KUKA KRL program: MyProgram_287().src

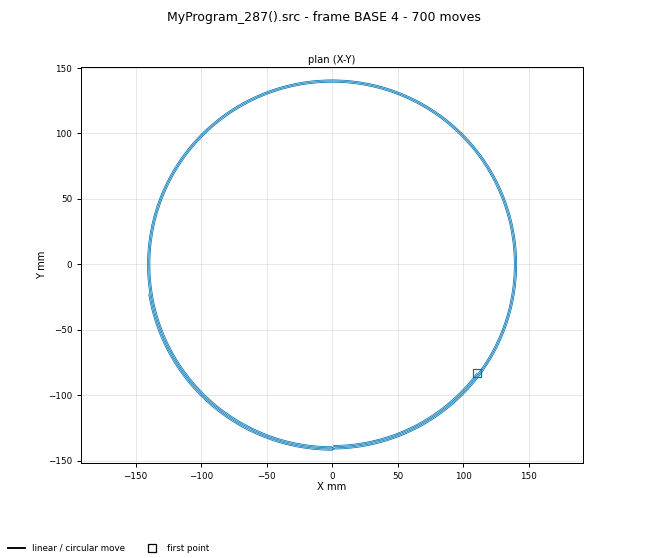
[picture p0: tool path of MyProgram_287().src in frame BASE 4, 700 of 700 moves have a stored position in this frame; points joined in program order, loops and branches not executed]
&ACCESS RVP
&REL 1
&PARAM TEMPLATE = C:\KRC\Roboter\Template\vorgabe
&PARAM EDITMASK = *
DEF MyProgram_287()
; ---- Setting reference (Base) ----
$BASE = BASE_DATA[4]

; --------------------------
; ---- Setting tool (TCP) ----
$TOOL = TOOL_DATA[3]
; --------------------------

$VEL.CP = VEL_APROX_PRINT
Startdeposition()
$VEL.CP = VEL_PRINT
LIN {X 110.6331,Y -82.8867,Z 175,A -34.5212,B 7.5627,C 0.3463,E1 7.6986,E2 486.4179} C_DIS
LIN {X 107.2416,Y -87.2299,Z 175,A -36.9213,B 7.5624,C 0.3539,E1 7.6944,E2 488.8351} C_DIS
LIN {X 102.8768,Y -92.3369,Z 175,A -39.3505,B 7.5624,C 0.3533,E1 7.69,E2 491.2213} C_DIS
LIN {X 98.1366,Y -97.3598,Z 175,A -42.4182,B 7.5619,C 0.3634,E1 7.6841,E2 494.3184} C_DIS
LIN {X 93.1713,Y -102.1223,Z 175,A -45.0279,B 7.5619,C 0.3647,E1 7.6789,E2 496.8996} C_DIS
LIN {X 87.5657,Y -106.9672,Z 175,A -48.9682,B 7.5608,C 0.3871,E1 7.6702,E2 500.9543} C_DIS
LIN {X 82.9444,Y -110.5898,Z 175,A -50.7968,B 7.5611,C 0.3802,E1 7.6663,E2 502.7077} C_DIS
LIN {X 78.2909,Y -113.9309,Z 175,A -53.0648,B 7.561,C 0.3823,E1 7.6611,E2 504.9642} C_DIS
LIN {X 74.3872,Y -116.5173,Z 175,A -54.9775,B 7.5609,C 0.3851,E1 7.6567,E2 506.8749} C_DIS
LIN {X 69.3615,Y -119.5773,Z 175,A -57.3901,B 7.5607,C 0.3884,E1 7.6509,E2 509.2862} C_DIS
LIN {X 65.5707,Y -121.6973,Z 175,A -59.228,B 7.5605,C 0.3918,E1 7.6464,E2 511.1304} C_DIS
LIN {X 61.8336,Y -123.6379,Z 175,A -60.9301,B 7.5605,C 0.3934,E1 7.6421,E2 512.8284} C_DIS
LIN {X 58.7912,Y -125.1139,Z 175,A -62.3873,B 7.5603,C 0.3963,E1 7.6385,E2 514.2939} C_DIS
LIN {X 53.8239,Y -127.3284,Z 175,A -64.525,B 7.5603,C 0.397,E1 7.633,E2 516.4183} C_DIS
LIN {X 49.8285,Y -128.9433,Z 175,A -66.4746,B 7.56,C 0.4021,E1 7.6279,E2 518.3903} C_DIS
LIN {X 45.7126,Y -130.4598,Z 175,A -68.0713,B 7.56,C 0.4001,E1 7.6238,E2 519.9599} C_DIS
LIN {X 41.2974,Y -131.9257,Z 175,A -70.0623,B 7.56,C 0.4031,E1 7.6184,E2 521.9604} C_DIS
LIN {X 37.6293,Y -133.0166,Z 175,A -71.3805,B 7.5601,C 0.3998,E1 7.615,E2 523.2451} C_DIS
LIN {X 34.2562,Y -133.9246,Z 175,A -73.2007,B 7.5597,C 0.4076,E1 7.6099,E2 525.1143} C_DIS
LIN {X 29.37,Y -135.0803,Z 175,A -75.02,B 7.5599,C 0.4046,E1 7.6051,E2 526.9012} C_DIS
LIN {X 26.0323,Y -135.7629,Z 175,A -76.4292,B 7.5599,C 0.4055,E1 7.6012,E2 528.3109} C_DIS
LIN {X 22.9559,Y -136.317,Z 175,A -78.4903,B 7.559,C 0.4196,E1 7.5953,E2 530.471} C_DIS
LIN {X 16.9955,Y -137.189,Z 175,A -80.2487,B 7.5597,C 0.408,E1 7.5907,E2 532.1364} C_DIS
LIN {X 13.2679,Y -137.5982,Z 175,A -81.6417,B 7.5597,C 0.4059,E1 7.5868,E2 533.5094} C_DIS
LIN {X 10.1361,Y -137.8643,Z 175,A -83.1514,B 7.5596,C 0.4099,E1 7.5826,E2 535.0465} C_DIS
LIN {X 5.4762,Y -138.128,Z 175,A -85.0409,B 7.5596,C 0.4096,E1 7.5773,E2 536.9311} C_DIS
LIN {X 1.0216,Y -138.2328,Z 175,A -86.8303,B 7.5596,C 0.409,E1 7.5723,E2 538.714} C_DIS
Enddeposition()
LIN {X 1.0216,Y -138.2328,Z 175,A -86.8303,B 7.5596,C 0.409,E1 7.5723,E2 538.714} C_DIS
Startdeposition()
$VEL.CP = VEL_PRINT
LIN {X 1.4201,Y -139.1373,Z 175,A -85.8495,B 7.508,C 0.3996,E1 7.5232,E2 537.6751} C_DIS
LIN {X 5.8285,Y -139.0214,Z 175,A -84.1991,B 7.5079,C 0.4021,E1 7.5277,E2 536.0455} C_DIS
LIN {X 9.2409,Y -138.8374,Z 175,A -82.6419,B 7.508,C 0.399,E1 7.5321,E2 534.4679} C_DIS
LIN {X 13.2856,Y -138.5071,Z 175,A -81.1056,B 7.508,C 0.4008,E1 7.5364,E2 532.9483} C_DIS
LIN {X 16.7511,Y -138.1311,Z 175,A -79.5636,B 7.508,C 0.3982,E1 7.5407,E2 531.3915} C_DIS
LIN {X 23.3229,Y -137.1748,Z 175,A -76.3997,B 7.5086,C 0.389,E1 7.5496,E2 528.1692} C_DIS
LIN {X 27.9525,Y -136.3062,Z 175,A -74.9929,B 7.5081,C 0.3973,E1 7.5532,E2 526.8316} C_DIS
LIN {X 35.5217,Y -134.5325,Z 175,A -72.0188,B 7.5081,C 0.3989,E1 7.5613,E2 523.8855} C_DIS
LIN {X 37.6917,Y -133.9405,Z 175,A -70.9319,B 7.5082,C 0.3951,E1 7.5642,E2 522.7769} C_DIS
LIN {X 41.1973,Y -132.9048,Z 175,A -69.4338,B 7.5083,C 0.3938,E1 7.5682,E2 521.2786} C_DIS
LIN {X 44.3172,Y -131.8968,Z 175,A -67.7638,B 7.5087,C 0.3866,E1 7.5728,E2 519.5654} C_DIS
LIN {X 47.5641,Y -130.761,Z 175,A -66.6566,B 7.5085,C 0.3908,E1 7.5756,E2 518.4981} C_DIS
LIN {X 51.0181,Y -129.4534,Z 175,A -65.0237,B 7.5087,C 0.3869,E1 7.5799,E2 516.8493} C_DIS
LIN {X 56.479,Y -127.1647,Z 175,A -62.7406,B 7.5087,C 0.3868,E1 7.5857,E2 514.5847} C_DIS
LIN {X 58.8003,Y -126.1084,Z 175,A -61.674,B 7.5087,C 0.3851,E1 7.5884,E2 513.5151} C_DIS
LIN {X 62.3508,Y -124.3934,Z 175,A -60.0875,B 7.5088,C 0.3836,E1 7.5924,E2 511.9322} C_DIS
LIN {X 65.2663,Y -122.8874,Z 175,A -58.7004,B 7.509,C 0.381,E1 7.5958,E2 510.5393} C_DIS
LIN {X 69.1818,Y -120.7274,Z 175,A -56.0217,B 7.5099,C 0.3623,E1 7.6026,E2 507.7481} C_DIS
LIN {X 74.9621,Y -117.2256,Z 175,A -54.2838,B 7.5091,C 0.3777,E1 7.6064,E2 506.1462} C_DIS
LIN {X 77.8365,Y -115.3373,Z 175,A -52.1354,B 7.5099,C 0.3613,E1 7.6116,E2 503.8999} C_DIS
LIN {X 82.166,Y -112.2942,Z 175,A -50.8362,B 7.5093,C 0.3743,E1 7.6143,E2 502.715} C_DIS
LIN {X 85.7474,Y -109.5838,Z 175,A -48.8324,B 7.5096,C 0.368,E1 7.6188,E2 500.6893} C_DIS
LIN {X 88.6836,Y -107.2212,Z 175,A -46.6577,B 7.5103,C 0.353,E1 7.6236,E2 498.4309} C_DIS
LIN {X 92.5552,Y -103.8977,Z 175,A -45.0634,B 7.5101,C 0.3586,E1 7.6268,E2 496.9018} C_DIS
LIN {X 95.9429,Y -100.7779,Z 175,A -43.2164,B 7.5102,C 0.3557,E1 7.6306,E2 495.0595} C_DIS
LIN {X 99.1505,Y -97.6238,Z 175,A -40.9161,B 7.5108,C 0.343,E1 7.6352,E2 492.6983} C_DIS
LIN {X 102.5453,Y -94.0513,Z 175,A -39.4326,B 7.5105,C 0.3493,E1 7.6379,E2 491.2849} C_DIS
LIN {X 106.3749,Y -89.6976,Z 175,A -37.3257,B 7.5105,C 0.3494,E1 7.6417,E2 489.2125} C_DIS
LIN {X 111.1691,Y -83.6817,Z 175,A -33.9616,B 7.511,C 0.3383,E1 7.6476,E2 485.8198} C_DIS
LIN {X 113.8489,Y -79.9979,Z 175,A -32.0815,B 7.5112,C 0.3337,E1 7.6506,E2 483.9372} C_DIS
LIN {X 116.2575,Y -76.455,Z 175,A -30.3464,B 7.5114,C 0.3299,E1 7.6533,E2 482.2042} C_DIS
LIN {X 119.2524,Y -71.6949,Z 175,A -28.1739,B 7.5115,C 0.327,E1 7.6565,E2 480.0482} C_DIS
LIN {X 121.1264,Y -68.4812,Z 175,A -26.5315,B 7.5118,C 0.3209,E1 7.6588,E2 478.3899} C_DIS
LIN {X 123.125,Y -64.814,Z 175,A -24.7076,B 7.512,C 0.3143,E1 7.6612,E2 476.5506} C_DIS
LIN {X 124.5929,Y -61.9468,Z 175,A -23.8146,B 7.5118,C 0.3195,E1 7.6622,E2 475.713} C_DIS
LIN {X 128.0502,Y -54.4463,Z 175,A -20.2779,B 7.5123,C 0.3078,E1 7.6664,E2 472.1556} C_DIS
LIN {X 129.844,Y -50.0134,Z 175,A -18.3416,B 7.5125,C 0.3031,E1 7.6683,E2 470.2216} C_DIS
LIN {X 130.9587,Y -47.0157,Z 175,A -17.0459,B 7.5126,C 0.2999,E1 7.6696,E2 468.9273} C_DIS
LIN {X 132.1846,Y -43.4529,Z 175,A -15.5767,B 7.5127,C 0.2973,E1 7.6709,E2 467.4674} C_DIS
LIN {X 133.6756,Y -38.6231,Z 175,A -13.2766,B 7.5131,C 0.2871,E1 7.6727,E2 465.1368} C_DIS
LIN {X 134.9715,Y -33.8161,Z 175,A -11.506,B 7.5131,C 0.287,E1 7.6739,E2 463.4006} C_DIS
LIN {X 135.7081,Y -30.7257,Z 175,A -10.2142,B 7.5133,C 0.2836,E1 7.6747,E2 462.1097} C_DIS
LIN {X 137.0688,Y -23.9412,Z 175,A -7.6666,B 7.5133,C 0.2816,E1 7.6761,E2 459.5988} C_DIS
LIN {X 137.6462,Y -20.3642,Z 175,A -6.0341,B 7.5136,C 0.2745,E1 7.6768,E2 457.9467} C_DIS
LIN {X 138.0565,Y -17.3679,Z 175,A -4.6261,B 7.5138,C 0.2677,E1 7.6773,E2 456.5165} C_DIS
LIN {X 138.7792,Y -10.0537,Z 175,A -1.8474,B 7.514,C 0.264,E1 7.678,E2 453.7672} C_DIS
LIN {X 138.9752,Y -6.8315,Z 175,A -0.4575,B 7.5141,C 0.2589,E1 7.6782,E2 452.3683} C_DIS
LIN {X 139.1026,Y -3.3845,Z 175,A 0.8979,B 7.5142,C 0.2561,E1 7.6784,E2 451.0201} C_DIS
LIN {X 139.1434,Y -0.4634,Z 175,A 2.037,B 7.5143,C 0.254,E1 7.6784,E2 449.8883} C_DIS
LIN {X 139.1107,Y 3.0949,Z 175,A 3.7076,B 7.5146,C 0.2456,E1 7.6784,E2 448.1898} C_DIS
LIN {X 138.8806,Y 8.5391,Z 175,A 5.8033,B 7.5147,C 0.2421,E1 7.678,E2 446.1113} C_DIS
LIN {X 138.5278,Y 13.0704,Z 175,A 8.0872,B 7.5151,C 0.2285,E1 7.6774,E2 443.7724} C_DIS
LIN {X 138.0155,Y 17.6805,Z 175,A 10.4809,B 7.5156,C 0.2133,E1 7.6765,E2 441.3139} C_DIS
LIN {X 136.852,Y 25.1523,Z 175,A 12.4644,B 7.5152,C 0.2272,E1 7.6757,E2 439.4752} C_DIS
LIN {X 135.5461,Y 31.4349,Z 175,A 15.0748,B 7.5154,C 0.2204,E1 7.6741,E2 436.867} C_DIS
LIN {X 134.6874,Y 34.9355,Z 175,A 16.5343,B 7.5154,C 0.2168,E1 7.6731,E2 435.4096} C_DIS
LIN {X 133.9536,Y 37.6448,Z 175,A 17.668,B 7.5155,C 0.214,E1 7.6723,E2 434.278} C_DIS
LIN {X 132.9674,Y 40.9925,Z 175,A 19.089,B 7.5157,C 0.2104,E1 7.6711,E2 432.8579} C_DIS
LIN {X 132.0076,Y 43.9844,Z 175,A 20.3873,B 7.5157,C 0.2068,E1 7.67,E2 431.5582} C_DIS
LIN {X 130.8447,Y 47.332,Z 175,A 21.8394,B 7.5159,C 0.203,E1 7.6686,E2 430.1061} C_DIS
LIN {X 129.5562,Y 50.7537,Z 175,A 23.2485,B 7.5159,C 0.2008,E1 7.6672,E2 428.7085} C_DIS
LIN {X 127.2737,Y 56.2354,Z 175,A 25.6984,B 7.5161,C 0.1943,E1 7.6646,E2 426.2565} C_DIS
LIN {X 125.0302,Y 61.0602,Z 175,A 27.7239,B 7.5161,C 0.1919,E1 7.6622,E2 424.2509} C_DIS
LIN {X 123.8823,Y 63.3549,Z 175,A 28.903,B 7.5163,C 0.1868,E1 7.6607,E2 423.0555} C_DIS
LIN {X 121.9898,Y 66.9311,Z 175,A 30.8976,B 7.5165,C 0.1762,E1 7.658,E2 421.018} C_DIS
LIN {X 120.1169,Y 70.2345,Z 175,A 32.4748,B 7.5166,C 0.172,E1 7.6557,E2 419.4382} C_DIS
LIN {X 117.9562,Y 73.808,Z 175,A 33.7508,B 7.5166,C 0.1765,E1 7.6539,E2 418.2183} C_DIS
LIN {X 115.7509,Y 77.2197,Z 175,A 35.2951,B 7.5166,C 0.175,E1 7.6516,E2 416.6896} C_DIS
LIN {X 113.7648,Y 80.1171,Z 175,A 36.9071,B 7.5167,C 0.1684,E1 7.649,E2 415.0558} C_DIS
LIN {X 110.9929,Y 83.9151,Z 175,A 39.2311,B 7.517,C 0.1565,E1 7.645,E2 412.6813} C_DIS
LIN {X 108.1615,Y 87.5345,Z 175,A 40.6057,B 7.5168,C 0.1622,E1 7.6427,E2 411.3722} C_DIS
LIN {X 105.5905,Y 90.6194,Z 175,A 42.3243,B 7.5169,C 0.1573,E1 7.6396,E2 409.6448} C_DIS
LIN {X 99.9105,Y 96.8455,Z 175,A 45.3488,B 7.5169,C 0.1585,E1 7.634,E2 406.6759} C_DIS
LIN {X 96.1312,Y 100.5973,Z 175,A 47.9075,B 7.5171,C 0.1472,E1 7.6288,E2 404.0703} C_DIS
LIN {X 93.3186,Y 103.2126,Z 175,A 49.4134,B 7.5171,C 0.1456,E1 7.6257,E2 402.5736} C_DIS
LIN {X 91.2332,Y 105.0608,Z 175,A 50.5802,B 7.5172,C 0.1431,E1 7.6233,E2 401.4041} C_DIS
LIN {X 87.8054,Y 107.942,Z 175,A 52.4091,B 7.5172,C 0.14,E1 7.6193,E2 399.5768} C_DIS
LIN {X 84.2147,Y 110.7664,Z 175,A 54.2717,B 7.5173,C 0.137,E1 7.6152,E2 397.7161} C_DIS
LIN {X 80.5882,Y 113.4322,Z 175,A 56.2153,B 7.5174,C 0.1323,E1 7.6108,E2 395.7609} C_DIS
LIN {X 75.6902,Y 116.7569,Z 175,A 58.3095,B 7.5174,C 0.1347,E1 7.606,E2 393.7099} C_DIS
LIN {X 72.5843,Y 118.7128,Z 175,A 59.9518,B 7.5174,C 0.13,E1 7.6021,E2 392.051} C_DIS
LIN {X 68.9617,Y 120.853,Z 175,A 61.7195,B 7.5175,C 0.1269,E1 7.5978,E2 390.2788} C_DIS
LIN {X 65.0323,Y 123.0104,Z 175,A 64.5964,B 7.5178,C 0.1057,E1 7.5904,E2 387.2703} C_DIS
LIN {X 57.7968,Y 126.5724,Z 175,A 66.851,B 7.5176,C 0.1209,E1 7.585,E2 385.152} C_DIS
LIN {X 51.8404,Y 129.1249,Z 175,A 69.4055,B 7.5176,C 0.12,E1 7.5785,E2 382.6122} C_DIS
LIN {X 48.426,Y 130.4443,Z 175,A 70.8827,B 7.5176,C 0.119,E1 7.5746,E2 381.139} C_DIS
LIN {X 44.9713,Y 131.6762,Z 175,A 72.3636,B 7.5176,C 0.1181,E1 7.5707,E2 379.6621} C_DIS
LIN {X 41.8074,Y 132.7143,Z 175,A 73.7259,B 7.5176,C 0.117,E1 7.5671,E2 378.301} C_DIS
LIN {X 38.8998,Y 133.5946,Z 175,A 75.0449,B 7.5177,C 0.1148,E1 7.5635,E2 376.9736} C_DIS
LIN {X 35.5899,Y 134.5143,Z 175,A 76.4451,B 7.5177,C 0.114,E1 7.5598,E2 375.5756} C_DIS
LIN {X 31.1855,Y 135.603,Z 175,A 78.2197,B 7.5177,C 0.1144,E1 7.555,E2 373.8132} C_DIS
LIN {X 24.6353,Y 136.9446,Z 175,A 80.7589,B 7.5177,C 0.1165,E1 7.5481,E2 371.3017} C_DIS
LIN {X 17.9569,Y 137.9793,Z 175,A 83.8373,B 7.5177,C 0.1103,E1 7.5395,E2 368.1873} C_DIS
LIN {X 13.5162,Y 138.485,Z 175,A 85.6921,B 7.5177,C 0.1095,E1 7.5344,E2 366.3314} C_DIS
LIN {X 9.3418,Y 138.8311,Z 175,A 87.5643,B 7.5178,C 0.1067,E1 7.5291,E2 364.4414} C_DIS
LIN {X 4.7477,Y 139.0636,Z 175,A 89.3336,B 7.5178,C 0.1085,E1 7.5242,E2 362.6886} C_DIS
LIN {X 0.3427,Y 139.1432,Z 175,A 91.0081,B 7.5178,C 0.1108,E1 7.5196,E2 361.0324} C_DIS
LIN {X -3.1295,Y 139.1097,Z 175,A 92.5251,B 7.5178,C 0.1094,E1 7.5153,E2 359.5052} C_DIS
LIN {X -9.7529,Y 138.8012,Z 175,A 95.0699,B 7.5178,C 0.1129,E1 7.5083,E2 356.985} C_DIS
LIN {X -16.5387,Y 138.1564,Z 175,A 98.0944,B 7.5178,C 0.1102,E1 7.4998,E2 353.9349} C_DIS
LIN {X -23.5222,Y 137.1415,Z 175,A 100.901,B 7.5178,C 0.113,E1 7.4921,E2 351.1425} C_DIS
LIN {X -26.4114,Y 136.6134,Z 175,A 102.1282,B 7.5178,C 0.1134,E1 7.4887,E2 349.9138} C_DIS
LIN {X -29.4419,Y 135.9921,Z 175,A 103.4486,B 7.5178,C 0.1134,E1 7.4851,E2 348.5883} C_DIS
LIN {X -33.1224,Y 135.1438,Z 175,A 105.0333,B 7.5178,C 0.114,E1 7.4808,E2 347.001} C_DIS
LIN {X -37.9549,Y 133.8668,Z 175,A 107.0155,B 7.5177,C 0.1167,E1 7.4755,E2 345.0297} C_DIS
LIN {X -41.1039,Y 132.9334,Z 175,A 108.3808,B 7.5177,C 0.1177,E1 7.4718,E2 343.6636} C_DIS
LIN {X -44.4666,Y 131.8471,Z 175,A 110.1098,B 7.5177,C 0.1147,E1 7.4671,E2 341.9013} C_DIS
LIN {X -50.2139,Y 129.7661,Z 175,A 112.5513,B 7.5177,C 0.1184,E1 7.4608,E2 339.4711} C_DIS
LIN {X -53.8552,Y 128.2977,Z 175,A 114.0667,B 7.5176,C 0.1218,E1 7.4569,E2 337.9696} C_DIS
LIN {X -57.3649,Y 126.7685,Z 175,A 116.1592,B 7.5176,C 0.1158,E1 7.4514,E2 335.8134} C_DIS
LIN {X -61.3669,Y 124.8789,Z 175,A 117.245,B 7.5175,C 0.1292,E1 7.4489,E2 334.8216} C_DIS
LIN {X -65.5803,Y 122.7212,Z 175,A 119.5789,B 7.5175,C 0.1261,E1 7.443,E2 332.4412} C_DIS
LIN {X -71.8801,Y 119.1404,Z 175,A 122.4019,B 7.5175,C 0.1328,E1 7.4363,E2 329.6409} C_DIS
LIN {X -75.9748,Y 116.5721,Z 175,A 124.5763,B 7.5175,C 0.1332,E1 7.4311,E2 327.445} C_DIS
LIN {X -79.8148,Y 113.9778,Z 175,A 126.5319,B 7.5174,C 0.1356,E1 7.4266,E2 325.4852} C_DIS
LIN {X -86.6506,Y 108.8707,Z 175,A 129.8564,B 7.5172,C 0.1445,E1 7.4192,E2 322.1877} C_DIS
LIN {X -89.3495,Y 106.6669,Z 175,A 131.5183,B 7.5172,C 0.1439,E1 7.4156,E2 320.4985} C_DIS
LIN {X -93.9561,Y 102.6328,Z 175,A 134.4308,B 7.5172,C 0.1431,E1 7.4094,E2 317.539} C_DIS
LIN {X -97.0129,Y 99.7485,Z 175,A 135.5603,B 7.517,C 0.1552,E1 7.4073,E2 316.4868} C_DIS
LIN {X -99.059,Y 97.7171,Z 175,A 137.0419,B 7.517,C 0.1534,E1 7.4043,E2 314.9693} C_DIS
LIN {X -103.493,Y 93.0077,Z 175,A 139.8811,B 7.517,C 0.1566,E1 7.3989,E2 312.1105} C_DIS
LIN {X -106.4377,Y 89.6228,Z 175,A 141.6227,B 7.5168,C 0.1622,E1 7.3958,E2 310.3841} C_DIS
LIN {X -109.2153,Y 86.2165,Z 175,A 143.5593,B 7.5168,C 0.1645,E1 7.3924,E2 308.4332} C_DIS
LIN {X -111.958,Y 82.6236,Z 175,A 145.2151,B 7.5166,C 0.1717,E1 7.3897,E2 306.8051} C_DIS
LIN {X -114.3086,Y 79.3394,Z 175,A 146.9862,B 7.5166,C 0.1741,E1 7.3868,E2 305.022} C_DIS
LIN {X -116.6391,Y 75.8715,Z 175,A 149.1485,B 7.5166,C 0.1721,E1 7.3834,E2 302.8054} C_DIS
LIN {X -118.9143,Y 72.254,Z 175,A 150.5098,B 7.5164,C 0.182,E1 7.3815,E2 301.4963} C_DIS
LIN {X -121.0516,Y 68.6136,Z 175,A 152.4285,B 7.5164,C 0.1839,E1 7.3788,E2 299.5564} C_DIS
LIN {X -123.3582,Y 64.3699,Z 175,A 154.2955,B 7.5162,C 0.1906,E1 7.3764,E2 297.7067} C_DIS
LIN {X -125.9505,Y 59.1418,Z 175,A 156.6895,B 7.516,C 0.197,E1 7.3734,E2 295.3164} C_DIS
LIN {X -127.1149,Y 56.5904,Z 175,A 157.8993,B 7.516,C 0.1993,E1 7.372,E2 294.1006} C_DIS
LIN {X -128.6045,Y 53.1206,Z 175,A 159.5168,B 7.5159,C 0.2026,E1 7.3703,E2 292.4767} C_DIS
LIN {X -129.7693,Y 50.2057,Z 175,A 160.8193,B 7.5158,C 0.2059,E1 7.369,E2 291.1742} C_DIS
LIN {X -131.0451,Y 46.7761,Z 175,A 162.3069,B 7.5157,C 0.2103,E1 7.3675,E2 289.6905} C_DIS
LIN {X -132.1799,Y 43.4669,Z 175,A 163.7712,B 7.5156,C 0.2139,E1 7.3662,E2 288.2247} C_DIS
LIN {X -133.1893,Y 40.2675,Z 175,A 165.176,B 7.5155,C 0.2174,E1 7.3651,E2 286.8181} C_DIS
LIN {X -134.0766,Y 37.2047,Z 175,A 166.4876,B 7.5153,C 0.2211,E1 7.3641,E2 285.5079} C_DIS
LIN {X -134.934,Y 33.9641,Z 175,A 167.9478,B 7.5153,C 0.2238,E1 7.3631,E2 284.039} C_DIS
LIN {X -135.7747,Y 30.434,Z 175,A 169.4504,B 7.5151,C 0.2279,E1 7.3621,E2 282.5367} C_DIS
LIN {X -137.0284,Y 24.1669,Z 175,A 172.0912,B 7.5149,C 0.2353,E1 7.3607,E2 279.8973} C_DIS
LIN {X -137.5307,Y 21.1194,Z 175,A 173.4536,B 7.5149,C 0.2377,E1 7.3601,E2 278.5245} C_DIS
LIN {X -138.0249,Y 17.6089,Z 175,A 174.9348,B 7.5147,C 0.2416,E1 7.3596,E2 277.042} C_DIS
LIN {X -138.6421,Y 11.794,Z 175,A 177.964,B 7.5147,C 0.24,E1 7.3588,E2 273.9355} C_DIS
LIN {X -138.9674,Y 6.9865,Z 175,A 179.1814,B 7.5142,C 0.2562,E1 7.3586,E2 272.8179} C_DIS
LIN {X -139.0886,Y 3.8883,Z 175,A -179.2932,B 7.5142,C 0.2565,E1 7.3584,E2 271.2621} C_DIS
LIN {X -139.1227,Y -2.3738,Z 175,A -176.2102,B 7.5142,C 0.257,E1 7.3584,E2 268.1167} C_DIS
LIN {X -138.9902,Y -6.5331,Z 175,A -174.9194,B 7.5138,C 0.2677,E1 7.3586,E2 266.8816} C_DIS
LIN {X -138.7817,Y -10.0191,Z 175,A -173.4204,B 7.5138,C 0.271,E1 7.3589,E2 265.376} C_DIS
LIN {X -137.9589,Y -18.1126,Z 175,A -170.291,B 7.5133,C 0.2836,E1 7.3598,E2 262.2777} C_DIS
LIN {X -137.5237,Y -21.1652,Z 175,A -168.7207,B 7.5133,C 0.2831,E1 7.3605,E2 260.6699} C_DIS
LIN {X -136.9491,Y -24.6097,Z 175,A -167.2575,B 7.5131,C 0.2868,E1 7.3612,E2 259.2047} C_DIS
LIN {X -136.3006,Y -27.9804,Z 175,A -165.787,B 7.5131,C 0.29,E1 7.362,E2 257.7279} C_DIS
LIN {X -135.5939,Y -31.2254,Z 175,A -164.4008,B 7.5129,C 0.2936,E1 7.3628,E2 256.3404} C_DIS
LIN {X -134.5408,Y -35.4905,Z 175,A -162.5242,B 7.5127,C 0.2977,E1 7.3641,E2 254.4564} C_DIS
LIN {X -133.5579,Y -39.0249,Z 175,A -161.0415,B 7.5125,C 0.3022,E1 7.3652,E2 252.9783} C_DIS
LIN {X -132.543,Y -42.3438,Z 175,A -159.5616,B 7.5125,C 0.3054,E1 7.3665,E2 251.4929} C_DIS
LIN {X -131.4827,Y -45.5295,Z 175,A -157.7465,B 7.5125,C 0.3031,E1 7.3682,E2 249.6228} C_DIS
LIN {X -130.0587,Y -49.4554,Z 175,A -156.0936,B 7.5123,C 0.3086,E1 7.3698,E2 247.9798} C_DIS
LIN {X -128.7403,Y -52.7943,Z 175,A -154.93,B 7.5119,C 0.3169,E1 7.371,E2 246.8578} C_DIS
LIN {X -127.5524,Y -55.5982,Z 175,A -153.654,B 7.5119,C 0.3199,E1 7.3724,E2 245.5796} C_DIS
LIN {X -126.0829,Y -58.8554,Z 175,A -152.1512,B 7.5117,C 0.3232,E1 7.3742,E2 244.0737} C_DIS
LIN {X -124.5708,Y -61.9916,Z 175,A -150.6623,B 7.5115,C 0.3261,E1 7.376,E2 242.5785} C_DIS
LIN {X -122.0654,Y -66.7924,Z 175,A -148.1366,B 7.5115,C 0.3275,E1 7.3794,E2 240.0158} C_DIS
LIN {X -120.4667,Y -69.6344,Z 175,A -147.0142,B 7.5112,C 0.3339,E1 7.3809,E2 238.9226} C_DIS
LIN {X -118.3216,Y -73.2208,Z 175,A -145.2045,B 7.5111,C 0.3368,E1 7.3835,E2 237.1022} C_DIS
LIN {X -115.8579,Y -77.0594,Z 175,A -143.4169,B 7.5108,C 0.3425,E1 7.3863,E2 235.3273} C_DIS
LIN {X -113.5757,Y -80.3851,Z 175,A -141.6366,B 7.5108,C 0.3446,E1 7.3891,E2 233.5323} C_DIS
LIN {X -110.862,Y -84.0886,Z 175,A -139.6983,B 7.5106,C 0.3482,E1 7.3924,E2 231.5886} C_DIS
LIN {X -108.1713,Y -87.5224,Z 175,A -137.8771,B 7.5104,C 0.3518,E1 7.3955,E2 229.7648} C_DIS
LIN {X -105.269,Y -90.9926,Z 175,A -135.2657,B 7.5107,C 0.3447,E1 7.4005,E2 227.0562} C_DIS
LIN {X -101.1736,Y -95.5252,Z 175,A -133.4924,B 7.51,C 0.3608,E1 7.4037,E2 225.3809} C_DIS
LIN {X -96.9244,Y -99.8342,Z 175,A -130.8928,B 7.5098,C 0.3641,E1 7.4088,E2 222.768} C_DIS
LIN {X -93.5684,Y -102.986,Z 175,A -128.9842,B 7.5096,C 0.3675,E1 7.4127,E2 220.8583} C_DIS
LIN {X -90.063,Y -106.0652,Z 175,A -127.0701,B 7.5095,C 0.371,E1 7.4168,E2 218.9455} C_DIS
LIN {X -86.7151,Y -108.8194,Z 175,A -125.2443,B 7.5093,C 0.3735,E1 7.4208,E2 217.1147} C_DIS
LIN {X -83.1111,Y -111.5961,Z 175,A -122.4545,B 7.5099,C 0.3625,E1 7.4273,E2 214.2047} C_DIS
LIN {X -77.3531,Y -115.6619,Z 175,A -120.7764,B 7.5087,C 0.3859,E1 7.4308,E2 212.6878} C_DIS
LIN {X -73.6761,Y -118.0383,Z 175,A -118.5713,B 7.5089,C 0.3823,E1 7.4361,E2 210.4304} C_DIS
LIN {X -69.7339,Y -120.4091,Z 175,A -116.6864,B 7.5088,C 0.385,E1 7.4406,E2 208.5468} C_DIS
LIN {X -61.2712,Y -124.9262,Z 175,A -112.7743,B 7.5085,C 0.3905,E1 7.4503,E2 204.6398} C_DIS
LIN {X -57.8945,Y -126.5272,Z 175,A -110.9833,B 7.5086,C 0.3882,E1 7.4549,E2 202.8157} C_DIS
LIN {X -53.3214,Y -128.5206,Z 175,A -109.131,B 7.5083,C 0.3935,E1 7.4596,E2 200.9897} C_DIS
LIN {X -50.1972,Y -129.7726,Z 175,A -107.7497,B 7.5083,C 0.3949,E1 7.4632,E2 199.6088} C_DIS
LIN {X -46.4865,Y -131.1495,Z 175,A -105.9915,B 7.5083,C 0.3943,E1 7.4679,E2 197.8336} C_DIS
LIN {X -42.3482,Y -132.5416,Z 175,A -104.2551,B 7.5082,C 0.3967,E1 7.4724,E2 196.1049} C_DIS
LIN {X -38.233,Y -133.7891,Z 175,A -102.1782,B 7.5084,C 0.3929,E1 7.4781,E2 193.9875} C_DIS
LIN {X -34.7328,Y -134.7389,Z 175,A -101.1637,B 7.5079,C 0.4017,E1 7.4807,E2 193.0355} C_DIS
LIN {X -29.4791,Y -135.9841,Z 175,A -98.8307,B 7.5079,C 0.4011,E1 7.4871,E2 190.6876} C_DIS
LIN {X -26.8383,Y -136.5318,Z 175,A -97.3699,B 7.5082,C 0.3957,E1 7.4912,E2 189.1805} C_DIS
LIN {X -23.4366,Y -137.1558,Z 175,A -96.1071,B 7.508,C 0.399,E1 7.4946,E2 187.9385} C_DIS
LIN {X -19.0966,Y -137.8274,Z 175,A -94.3386,B 7.508,C 0.4002,E1 7.4995,E2 186.1746} C_DIS
LIN {X -15.1435,Y -138.3165,Z 175,A -92.8275,B 7.5078,C 0.4027,E1 7.5037,E2 184.6799} C_DIS
LIN {X -11.7404,Y -138.6467,Z 175,A -91.3654,B 7.5078,C 0.402,E1 7.5077,E2 183.2101} C_DIS
LIN {X -7.9854,Y -138.9147,Z 175,A -89.8713,B 7.5078,C 0.403,E1 7.5119,E2 181.7228} C_DIS
LIN {X -4.0978,Y -139.0828,Z 175,A -88.2235,B 7.5078,C 0.4022,E1 7.5165,E2 180.0683} C_DIS
LIN {X -0.5851,Y -139.1419,Z 175,A -86.7915,B 7.5078,C 0.4023,E1 7.5205,E2 178.6374} C_DIS
LIN {X -0.5851,Y -139.1419,Z 175,A -86.7915,B 7.5078,C 0.4023,E1 7.5205,E2 178.6374} C_DIS
Enddeposition()
LIN {X 1.0319,Y -140.0436,Z 175,A -86.268,B 7.3266,C 0.4098,E1 7.3411,E2 178.2178} C_DIS
Startdeposition()
$VEL.CP = VEL_PRINT
LIN {X -1.9507,Y -140.0364,Z 175,A -87.9285,B 7.3262,C 0.4173,E1 7.3363,E2 179.937} C_DIS
LIN {X -5.5457,Y -139.9396,Z 175,A -89.3774,B 7.3262,C 0.417,E1 7.3322,E2 181.3836} C_DIS
LIN {X -9.8632,Y -139.702,Z 175,A -91.1972,B 7.3262,C 0.4177,E1 7.3271,E2 183.2108} C_DIS
LIN {X -13.6059,Y -139.387,Z 175,A -92.7276,B 7.3262,C 0.4174,E1 7.3229,E2 184.741} C_DIS
LIN {X -18.1814,Y -138.8641,Z 175,A -94.5962,B 7.3262,C 0.4167,E1 7.3177,E2 186.6082} C_DIS
LIN {X -21.944,Y -138.3204,Z 175,A -96.4481,B 7.326,C 0.4211,E1 7.3125,E2 188.4994} C_DIS
LIN {X -25.5413,Y -137.7024,Z 175,A -97.565,B 7.3264,C 0.4144,E1 7.3096,E2 189.5676} C_DIS
LIN {X -29.3817,Y -136.9325,Z 175,A -99.6061,B 7.326,C 0.4207,E1 7.3038,E2 191.6664} C_DIS
LIN {X -33.1759,Y -136.0634,Z 175,A -100.829,B 7.3264,C 0.4139,E1 7.3006,E2 192.8415} C_DIS
LIN {X -38.8873,Y -134.5427,Z 175,A -103.107,B 7.3266,C 0.4101,E1 7.2945,E2 195.1018} C_DIS
LIN {X -42.8551,Y -133.3313,Z 175,A -104.9633,B 7.3266,C 0.4114,E1 7.2895,E2 196.9793} C_DIS
LIN {X -46.5618,Y -132.0843,Z 175,A -106.5583,B 7.3266,C 0.41,E1 7.2853,E2 198.574} C_DIS
LIN {X -49.3961,Y -131.0489,Z 175,A -107.7624,B 7.3267,C 0.4084,E1 7.2822,E2 199.7742} C_DIS
LIN {X -52.5844,Y -129.8023,Z 175,A -109.2141,B 7.3267,C 0.4079,E1 7.2784,E2 201.2328} C_DIS
LIN {X -56.3031,Y -128.2353,Z 175,A -111.2013,B 7.3265,C 0.4114,E1 7.2732,E2 203.264} C_DIS
LIN {X -59.5108,Y -126.7785,Z 175,A -112.309,B 7.3269,C 0.4047,E1 7.2705,E2 204.3283} C_DIS
LIN {X -68.4137,Y -122.2042,Z 175,A -116.5277,B 7.3271,C 0.4016,E1 7.26,E2 208.5634} C_DIS
LIN {X -72.1901,Y -120.0123,Z 175,A -118.3502,B 7.3271,C 0.3997,E1 7.2556,E2 210.3906} C_DIS
LIN {X -76.4269,Y -117.3594,Z 175,A -120.2085,B 7.3275,C 0.3939,E1 7.2513,E2 212.2244} C_DIS
LIN {X -79.3886,Y -115.3765,Z 175,A -122.3589,B 7.3271,C 0.4019,E1 7.2461,E2 214.4644} C_DIS
LIN {X -83.2986,Y -112.5867,Z 175,A -123.7949,B 7.3277,C 0.391,E1 7.243,E2 215.8318} C_DIS
LIN {X -86.351,Y -110.2623,Z 175,A -125.4657,B 7.3277,C 0.3898,E1 7.2393,E2 217.5155} C_DIS
LIN {X -89.831,Y -107.4462,Z 175,A -127.3441,B 7.3279,C 0.3873,E1 7.2352,E2 219.3996} C_DIS
LIN {X -93.226,Y -104.5143,Z 175,A -129.2076,B 7.328,C 0.3844,E1 7.2313,E2 221.2664} C_DIS
LIN {X -96.6181,Y -101.3866,Z 175,A -131.5524,B 7.3278,C 0.3874,E1 7.2265,E2 223.6697} C_DIS
LIN {X -99.9767,Y -98.076,Z 175,A -132.8445,B 7.3285,C 0.3745,E1 7.2241,E2 224.879} C_DIS
LIN {X -106.1203,Y -91.3933,Z 175,A -136.7981,B 7.3287,C 0.3703,E1 7.2166,E2 228.8626} C_DIS
LIN {X -108.8914,Y -88.0735,Z 175,A -138.6089,B 7.3289,C 0.3671,E1 7.2134,E2 230.6781} C_DIS
LIN {X -111.6105,Y -84.6016,Z 175,A -140.4178,B 7.3291,C 0.3631,E1 7.2103,E2 232.487} C_DIS
LIN {X -114.2013,Y -81.0709,Z 175,A -142.2602,B 7.3292,C 0.3598,E1 7.2073,E2 234.3352} C_DIS
LIN {X -116.7381,Y -77.3735,Z 175,A -144.1571,B 7.3294,C 0.3563,E1 7.2043,E2 236.2392} C_DIS
LIN {X -118.6054,Y -74.4789,Z 175,A -145.4767,B 7.3296,C 0.3518,E1 7.2023,E2 237.5466} C_DIS
LIN {X -121.214,Y -70.1527,Z 175,A -148.4045,B 7.3293,C 0.3585,E1 7.1981,E2 240.5835} C_DIS
LIN {X -124.1764,Y -64.7616,Z 175,A -150.1388,B 7.3301,C 0.3416,E1 7.1959,E2 242.2165} C_DIS
LIN {X -125.7633,Y -61.6232,Z 175,A -151.6064,B 7.3303,C 0.3383,E1 7.1941,E2 243.6871} C_DIS
LIN {X -127.3125,Y -58.3562,Z 175,A -153.105,B 7.3304,C 0.3348,E1 7.1923,E2 245.1873} C_DIS
LIN {X -128.9412,Y -54.6666,Z 175,A -155.0577,B 7.3304,C 0.3346,E1 7.1901,E2 247.1779} C_DIS
LIN {X -130.5953,Y -50.5826,Z 175,A -156.6012,B 7.3308,C 0.3263,E1 7.1885,E2 248.687} C_DIS
LIN {X -132.2093,Y -46.2011,Z 175,A -158.3776,B 7.3311,C 0.3194,E1 7.1869,E2 250.4449} C_DIS
LIN {X -132.9667,Y -43.9733,Z 175,A -159.5955,B 7.3311,C 0.3202,E1 7.1858,E2 251.695} C_DIS
LIN {X -134.1266,Y -40.3024,Z 175,A -161.2982,B 7.3311,C 0.3177,E1 7.1843,E2 253.413} C_DIS
LIN {X -135.298,Y -36.1691,Z 175,A -163.0008,B 7.3314,C 0.3121,E1 7.1831,E2 255.1073} C_DIS
LIN {X -136.257,Y -32.3729,Z 175,A -164.5786,B 7.3316,C 0.3073,E1 7.182,E2 256.6808} C_DIS
LIN {X -137.1386,Y -28.408,Z 175,A -166.3526,B 7.3318,C 0.3042,E1 7.181,E2 258.468} C_DIS
LIN {X -137.8753,Y -24.58,Z 175,A -167.9159,B 7.332,C 0.2993,E1 7.1802,E2 260.0261} C_DIS
LIN {X -138.4903,Y -20.8466,Z 175,A -169.642,B 7.332,C 0.2972,E1 7.1794,E2 261.7737} C_DIS
LIN {X -139.4034,Y -13.4356,Z 175,A -172.7002,B 7.3324,C 0.2886,E1 7.1785,E2 264.8299} C_DIS
LIN {X -139.7099,Y -9.7553,Z 175,A -174.469,B 7.3324,C 0.2876,E1 7.1781,E2 266.6301} C_DIS
LIN {X -139.9089,Y -6.2805,Z 175,A -175.7802,B 7.3326,C 0.2821,E1 7.1779,E2 267.9259} C_DIS
LIN {X -140.0215,Y 2.8459,Z 175,A -179.2729,B 7.3331,C 0.2682,E1 7.1779,E2 271.3849} C_DIS
LIN {X -139.8357,Y 7.7239,Z 175,A 178.3432,B 7.3331,C 0.2675,E1 7.1782,E2 273.8161} C_DIS
LIN {X -139.0685,Y 16.546,Z 175,A 175.1028,B 7.3337,C 0.2521,E1 7.179,E2 277.0048} C_DIS
LIN {X -138.675,Y 19.5727,Z 175,A 173.2451,B 7.3336,C 0.2565,E1 7.1797,E2 278.9385} C_DIS
LIN {X -138.1342,Y 23.0806,Z 175,A 172.2846,B 7.3339,C 0.246,E1 7.1801,E2 279.8356} C_DIS
LIN {X -137.3674,Y 27.2839,Z 175,A 170.3377,B 7.334,C 0.2436,E1 7.1811,E2 281.8061} C_DIS
LIN {X -136.5234,Y 31.227,Z 175,A 168.6226,B 7.3341,C 0.2398,E1 7.1822,E2 283.528} C_DIS
LIN {X -135.6512,Y 34.823,Z 175,A 167.1145,B 7.3343,C 0.2355,E1 7.1832,E2 285.0339} C_DIS
LIN {X -134.8398,Y 37.8415,Z 175,A 165.7942,B 7.3343,C 0.2325,E1 7.1842,E2 286.3583} C_DIS
LIN {X -133.8809,Y 41.1053,Z 175,A 164.3501,B 7.3345,C 0.2294,E1 7.1853,E2 287.8077} C_DIS
LIN {X -132.8375,Y 44.3616,Z 175,A 162.9181,B 7.3345,C 0.2259,E1 7.1866,E2 289.2425} C_DIS
LIN {X -131.4791,Y 48.245,Z 175,A 161.2323,B 7.3347,C 0.2214,E1 7.1882,E2 290.9271} C_DIS
LIN {X -130.3037,Y 51.3327,Z 175,A 159.8718,B 7.3348,C 0.2179,E1 7.1895,E2 292.2874} C_DIS
LIN {X -129.3067,Y 53.7914,Z 175,A 158.6963,B 7.3348,C 0.2162,E1 7.1908,E2 293.4732} C_DIS
LIN {X -127.7975,Y 57.2844,Z 175,A 156.8645,B 7.3348,C 0.2157,E1 7.1929,E2 295.338} C_DIS
LIN {X -126.4024,Y 60.3003,Z 175,A 155.6807,B 7.335,C 0.2098,E1 7.1943,E2 296.4984} C_DIS
LIN {X -124.6036,Y 63.9362,Z 175,A 154.0883,B 7.3352,C 0.2046,E1 7.1963,E2 298.0808} C_DIS
LIN {X -122.891,Y 67.172,Z 175,A 152.3527,B 7.3352,C 0.204,E1 7.1986,E2 299.8448} C_DIS
LIN {X -121.0564,Y 70.4251,Z 175,A 150.8905,B 7.3353,C 0.1993,E1 7.2006,E2 301.2975} C_DIS
LIN {X -117.4755,Y 76.248,Z 175,A 148.0992,B 7.3355,C 0.1924,E1 7.2048,E2 304.0854} C_DIS
LIN {X -115.1616,Y 79.7005,Z 175,A 146.3092,B 7.3355,C 0.1895,E1 7.2076,E2 305.885} C_DIS
LIN {X -112.5853,Y 83.3005,Z 175,A 144.3253,B 7.3356,C 0.1876,E1 7.2109,E2 307.8888} C_DIS
LIN {X -109.869,Y 86.8518,Z 175,A 142.8067,B 7.3358,C 0.1793,E1 7.2134,E2 309.3668} C_DIS
LIN {X -107.6796,Y 89.5513,Z 175,A 140.7283,B 7.3358,C 0.185,E1 7.2173,E2 311.5258} C_DIS
LIN {X -104.5735,Y 93.1599,Z 175,A 138.5482,B 7.3358,C 0.1839,E1 7.2214,E2 313.7328} C_DIS
LIN {X -100.6118,Y 97.4244,Z 175,A 136.9425,B 7.3361,C 0.1684,E1 7.2243,E2 315.2399} C_DIS
LIN {X -94.9987,Y 102.9057,Z 175,A 132.909,B 7.336,C 0.1733,E1 7.2327,E2 319.3729} C_DIS
LIN {X -90.7654,Y 106.6578,Z 175,A 131.1944,B 7.3363,C 0.1607,E1 7.2361,E2 321.0111} C_DIS
LIN {X -85.4296,Y 110.9772,Z 175,A 128.1807,B 7.3363,C 0.1585,E1 7.2428,E2 324.0479} C_DIS
LIN {X -82.8653,Y 112.9052,Z 175,A 127.0643,B 7.3364,C 0.1535,E1 7.2452,E2 325.1387} C_DIS
LIN {X -79.3834,Y 115.38,Z 175,A 125.255,B 7.3364,C 0.1515,E1 7.2494,E2 326.9542} C_DIS
LIN {X -75.3394,Y 118.0605,Z 175,A 123.3152,B 7.3365,C 0.1477,E1 7.2539,E2 328.8867} C_DIS
LIN {X -71.794,Y 120.2493,Z 175,A 121.1702,B 7.3365,C 0.1515,E1 7.2591,E2 331.0851} C_DIS
LIN {X -68.1513,Y 122.351,Z 175,A 119.8681,B 7.3366,C 0.143,E1 7.2622,E2 332.3339} C_DIS
LIN {X -64.8167,Y 124.1474,Z 175,A 118.3188,B 7.3366,C 0.1409,E1 7.266,E2 333.8818} C_DIS
LIN {X -61.5633,Y 125.7928,Z 175,A 116.0031,B 7.3365,C 0.151,E1 7.2721,E2 336.2985} C_DIS
LIN {X -55.9869,Y 128.372,Z 175,A 114.433,B 7.3368,C 0.1342,E1 7.2758,E2 337.7498} C_DIS
LIN {X -50.6049,Y 130.5866,Z 175,A 112.0727,B 7.3368,C 0.1314,E1 7.2819,E2 340.1059} C_DIS
LIN {X -45.3637,Y 132.4996,Z 175,A 109.6304,B 7.3368,C 0.1315,E1 7.2883,E2 342.5666} C_DIS
LIN {X -42.3028,Y 133.5077,Z 175,A 108.2387,B 7.3368,C 0.1315,E1 7.292,E2 343.9665} C_DIS
LIN {X -38.1267,Y 134.7601,Z 175,A 106.3652,B 7.3368,C 0.1314,E1 7.2971,E2 345.8501} C_DIS
LIN {X -34.3294,Y 135.7765,Z 175,A 104.845,B 7.3368,C 0.1289,E1 7.3012,E2 347.3582} C_DIS
LIN {X -30.4304,Y 136.7053,Z 175,A 103.002,B 7.3368,C 0.1309,E1 7.3062,E2 349.2256} C_DIS
LIN {X -25.8818,Y 137.6375,Z 175,A 101.3351,B 7.3369,C 0.1263,E1 7.3107,E2 350.8623} C_DIS
LIN {X -19.725,Y 138.6533,Z 175,A 98.7567,B 7.3369,C 0.1256,E1 7.3179,E2 353.4425} C_DIS
LIN {X -16.6202,Y 139.0596,Z 175,A 97.39,B 7.3369,C 0.1264,E1 7.3217,E2 354.8192} C_DIS
LIN {X -10.7126,Y 139.64,Z 175,A 94.9738,B 7.3369,C 0.1256,E1 7.3284,E2 357.2326} C_DIS
LIN {X -5.6476,Y 139.9356,Z 175,A 92.9298,B 7.3369,C 0.1248,E1 7.3341,E2 359.2716} C_DIS
LIN {X -1.7021,Y 140.0405,Z 175,A 91.227,B 7.3369,C 0.1261,E1 7.3388,E2 360.9847} C_DIS
LIN {X 2.1192,Y 140.0336,Z 175,A 89.6057,B 7.3369,C 0.1271,E1 7.3434,E2 362.6125} C_DIS
LIN {X 6.0096,Y 139.9215,Z 175,A 87.9821,B 7.3369,C 0.1278,E1 7.3479,E2 364.2393} C_DIS
LIN {X 11.0055,Y 139.6184,Z 175,A 86.15,B 7.3369,C 0.1247,E1 7.353,E2 366.0438} C_DIS
LIN {X 14.2705,Y 139.3222,Z 175,A 84.6557,B 7.3369,C 0.1276,E1 7.3572,E2 367.5567} C_DIS
LIN {X 19.0033,Y 138.7555,Z 175,A 82.4639,B 7.3369,C 0.1323,E1 7.3633,E2 369.778} C_DIS
LIN {X 22.6688,Y 138.203,Z 175,A 81.3057,B 7.3369,C 0.1271,E1 7.3664,E2 370.891} C_DIS
LIN {X 26.4444,Y 137.53,Z 175,A 79.6449,B 7.3369,C 0.1294,E1 7.371,E2 372.5628} C_DIS
LIN {X 30.4834,Y 136.6932,Z 175,A 78.0054,B 7.3369,C 0.1296,E1 7.3754,E2 374.1959} C_DIS
LIN {X 34.497,Y 135.734,Z 175,A 76.3494,B 7.3369,C 0.1303,E1 7.3799,E2 375.8475} C_DIS
LIN {X 38.839,Y 134.5569,Z 175,A 74.4983,B 7.3369,C 0.1319,E1 7.3849,E2 377.6995} C_DIS
LIN {X 42.6409,Y 133.3997,Z 175,A 72.9389,B 7.3369,C 0.1321,E1 7.389,E2 379.2503} C_DIS
LIN {X 46.2011,Y 132.2093,Z 175,A 71.4679,B 7.3369,C 0.1324,E1 7.3929,E2 380.7129} C_DIS
LIN {X 49.3913,Y 131.0507,Z 175,A 70.0372,B 7.3368,C 0.1345,E1 7.3967,E2 382.1488} C_DIS
LIN {X 52.5394,Y 129.8205,Z 175,A 68.2994,B 7.3367,C 0.1421,E1 7.4013,E2 383.9308} C_DIS
LIN {X 56.1274,Y 128.3112,Z 175,A 67.1142,B 7.3367,C 0.1369,E1 7.4042,E2 385.0649} C_DIS
LIN {X 59.0456,Y 126.9937,Z 175,A 65.1323,B 7.3365,C 0.1501,E1 7.4094,E2 387.1306} C_DIS
LIN {X 63.9241,Y 124.6097,Z 175,A 63.5491,B 7.3367,C 0.1419,E1 7.4132,E2 388.6343} C_DIS
LIN {X 67.9537,Y 122.4605,Z 175,A 61.6882,B 7.3367,C 0.1443,E1 7.4177,E2 390.4943} C_DIS
LIN {X 71.8194,Y 120.2341,Z 175,A 59.8188,B 7.3365,C 0.1478,E1 7.4222,E2 392.3693} C_DIS
LIN {X 75.5942,Y 117.8973,Z 175,A 58.0746,B 7.3365,C 0.1493,E1 7.4264,E2 394.1046} C_DIS
LIN {X 80.7057,Y 114.4589,Z 175,A 55.5542,B 7.3365,C 0.1533,E1 7.4322,E2 396.6252} C_DIS
LIN {X 84.1802,Y 111.9285,Z 175,A 53.8356,B 7.3364,C 0.1556,E1 7.436,E2 398.3391} C_DIS
LIN {X 87.6871,Y 109.203,Z 175,A 51.9913,B 7.3364,C 0.1593,E1 7.4401,E2 400.1872} C_DIS
LIN {X 91.1427,Y 106.3361,Z 175,A 50.1756,B 7.3362,C 0.1624,E1 7.4439,E2 402.0006} C_DIS
LIN {X 94.6518,Y 103.2244,Z 175,A 47.9004,B 7.336,C 0.1725,E1 7.4487,E2 404.3209} C_DIS
LIN {X 97.9608,Y 100.0897,Z 175,A 46.5095,B 7.3361,C 0.1676,E1 7.4514,E2 405.6529} C_DIS
LIN {X 100.9663,Y 97.0578,Z 175,A 44.7363,B 7.3361,C 0.1717,E1 7.4549,E2 407.4299} C_DIS
LIN {X 104.9147,Y 92.7747,Z 175,A 42.5257,B 7.336,C 0.1735,E1 7.459,E2 409.6194} C_DIS
LIN {X 107.3607,Y 89.933,Z 175,A 40.5381,B 7.3357,C 0.1853,E1 7.4627,E2 411.6649} C_DIS
LIN {X 110.0059,Y 86.6766,Z 175,A 39.1682,B 7.3357,C 0.1827,E1 7.465,E2 412.9917} C_DIS
LIN {X 112.4401,Y 83.4955,Z 175,A 37.5938,B 7.3357,C 0.1852,E1 7.4676,E2 414.5587} C_DIS
LIN {X 115.1288,Y 79.7477,Z 175,A 35.6898,B 7.3356,C 0.19,E1 7.4707,E2 416.4656} C_DIS
LIN {X 117.5673,Y 76.1066,Z 175,A 33.9717,B 7.3356,C 0.1928,E1 7.4733,E2 418.1751} C_DIS
LIN {X 119.9981,Y 72.2135,Z 175,A 31.6283,B 7.3351,C 0.2062,E1 7.4768,E2 420.5782} C_DIS
LIN {X 122.4968,Y 67.888,Z 175,A 30.2679,B 7.3354,C 0.1984,E1 7.4785,E2 421.8532} C_DIS
LIN {X 124.1749,Y 64.7643,Z 175,A 28.7768,B 7.3352,C 0.2028,E1 7.4805,E2 423.3502} C_DIS
LIN {X 125.6796,Y 61.7929,Z 175,A 27.0833,B 7.335,C 0.2126,E1 7.4826,E2 425.0865} C_DIS
LIN {X 127.3002,Y 58.3828,Z 175,A 26.0293,B 7.3351,C 0.2073,E1 7.4838,E2 426.079} C_DIS
LIN {X 129.9469,Y 52.2258,Z 175,A 23.5884,B 7.3351,C 0.2087,E1 7.4865,E2 428.4831} C_DIS
LIN {X 131.2565,Y 48.842,Z 175,A 21.7541,B 7.3348,C 0.2194,E1 7.4883,E2 430.3632} C_DIS
LIN {X 132.4509,Y 45.5043,Z 175,A 20.3151,B 7.3347,C 0.2231,E1 7.4897,E2 431.8017} C_DIS
LIN {X 133.5955,Y 42.028,Z 175,A 18.9221,B 7.3346,C 0.2252,E1 7.4908,E2 433.1825} C_DIS
LIN {X 134.374,Y 39.4638,Z 175,A 17.8017,B 7.3345,C 0.2287,E1 7.4917,E2 434.3067} C_DIS
LIN {X 135.3688,Y 35.9036,Z 175,A 16.306,B 7.3344,C 0.2325,E1 7.4928,E2 435.8013} C_DIS
LIN {X 136.3834,Y 31.8397,Z 175,A 14.6335,B 7.3342,C 0.2365,E1 7.4939,E2 437.4698} C_DIS
LIN {X 137.0669,Y 28.7594,Z 175,A 13.3855,B 7.3342,C 0.2393,E1 7.4947,E2 438.7133} C_DIS
LIN {X 137.6876,Y 25.6197,Z 175,A 12.0877,B 7.334,C 0.2428,E1 7.4954,E2 440.0106} C_DIS
LIN {X 138.3406,Y 21.8132,Z 175,A 9.9832,B 7.3335,C 0.2574,E1 7.4963,E2 442.1833} C_DIS
LIN {X 139.0146,Y 16.9977,Z 175,A 8.3612,B 7.3335,C 0.256,E1 7.4969,E2 443.76} C_DIS
LIN {X 139.4364,Y 13.0916,Z 175,A 6.9658,B 7.3335,C 0.2564,E1 7.4972,E2 445.1296} C_DIS
LIN {X 139.7688,Y 8.8652,Z 175,A 5.2659,B 7.3335,C 0.2607,E1 7.4976,E2 446.8263} C_DIS
LIN {X 139.9945,Y 3.9228,Z 175,A 3.4351,B 7.3333,C 0.2628,E1 7.4978,E2 448.634} C_DIS
LIN {X 140.049,Y 0.6188,Z 175,A 1.9686,B 7.3331,C 0.2689,E1 7.4978,E2 450.1164} C_DIS
LIN {X 139.9986,Y -3.7752,Z 175,A 0.2133,B 7.333,C 0.2732,E1 7.4978,E2 451.8678} C_DIS
LIN {X 139.8659,Y -7.1686,Z 175,A -1.1351,B 7.3328,C 0.2764,E1 7.4976,E2 453.2122} C_DIS
LIN {X 139.3539,Y -13.9515,Z 175,A -3.7956,B 7.3326,C 0.2821,E1 7.497,E2 455.8593} C_DIS
LIN {X 139.0209,Y -16.9446,Z 175,A -5.0668,B 7.3325,C 0.2864,E1 7.4966,E2 457.1367} C_DIS
LIN {X 138.5229,Y -20.6353,Z 175,A -6.6454,B 7.3323,C 0.2918,E1 7.4959,E2 458.7239} C_DIS
LIN {X 137.8031,Y -24.9838,Z 175,A -8.6095,B 7.3319,C 0.3001,E1 7.495,E2 460.7103} C_DIS
LIN {X 137.1673,Y -28.2669,Z 175,A -9.6245,B 7.332,C 0.297,E1 7.4945,E2 461.681} C_DIS
LIN {X 136.6061,Y -30.865,Z 175,A -11.0138,B 7.3317,C 0.306,E1 7.4936,E2 463.1104} C_DIS
LIN {X 135.8369,Y -34.091,Z 175,A -12.1143,B 7.3317,C 0.3048,E1 7.4929,E2 464.1791} C_DIS
LIN {X 134.2284,Y -39.9609,Z 175,A -14.5609,B 7.3315,C 0.3109,E1 7.491,E2 466.6224} C_DIS
LIN {X 133.2231,Y -43.1937,Z 175,A -15.8358,B 7.3314,C 0.3126,E1 7.4899,E2 467.8844} C_DIS
LIN {X 132.0265,Y -46.7269,Z 175,A -17.6543,B 7.331,C 0.3225,E1 7.4882,E2 469.7422} C_DIS
LIN {X 130.8634,Y -49.8914,Z 175,A -18.7164,B 7.331,C 0.3201,E1 7.4872,E2 470.7646} C_DIS
LIN {X 129.7374,Y -52.7454,Z 175,A -20.0431,B 7.3309,C 0.3249,E1 7.4858,E2 472.1018} C_DIS
LIN {X 127.8825,Y -57.0945,Z 175,A -22.2404,B 7.3304,C 0.3351,E1 7.4833,E2 474.335} C_DIS
LIN {X 126.213,Y -60.6967,Z 175,A -23.0763,B 7.3309,C 0.3241,E1 7.4825,E2 475.0699} C_DIS
LIN {X 124.8382,Y -63.4753,Z 175,A -24.6799,B 7.3305,C 0.334,E1 7.4804,E2 476.7186} C_DIS
LIN {X 123.2759,Y -66.4631,Z 175,A -26.1308,B 7.3302,C 0.3389,E1 7.4785,E2 478.1802} C_DIS
LIN {X 121.1842,Y -70.2043,Z 175,A -27.8389,B 7.3301,C 0.3425,E1 7.4761,E2 479.8841} C_DIS
LIN {X 118.5407,Y -74.5811,Z 175,A -29.8831,B 7.3299,C 0.3468,E1 7.4731,E2 481.9242} C_DIS
LIN {X 116.326,Y -77.9909,Z 175,A -31.5517,B 7.3297,C 0.351,E1 7.4706,E2 483.595} C_DIS
LIN {X 113.0687,Y -82.6427,Z 175,A -33.754,B 7.3295,C 0.3542,E1 7.467,E2 485.7839} C_DIS
LIN {X 109.1824,Y -87.7127,Z 175,A -36.364,B 7.3292,C 0.3603,E1 7.4626,E2 488.396} C_DIS
LIN {X 106.5902,Y -90.8449,Z 175,A -38.0349,B 7.329,C 0.3642,E1 7.4596,E2 490.0695} C_DIS
LIN {X 102.6134,Y -95.3141,Z 175,A -40.6038,B 7.3286,C 0.3719,E1 7.4547,E2 492.6565} C_DIS
LIN {X 99.103,Y -98.9594,Z 175,A -42.4499,B 7.3286,C 0.372,E1 7.4512,E2 494.4753} C_DIS
LIN {X 96.2104,Y -101.7734,Z 175,A -44.0684,B 7.3285,C 0.3748,E1 7.4479,E2 496.0911} C_DIS
LIN {X 92.5586,Y -105.1058,Z 175,A -46.3016,B 7.3281,C 0.3828,E1 7.4432,E2 498.3537} C_DIS
LIN {X 90.0963,Y -107.2237,Z 175,A -47.1689,B 7.3284,C 0.3768,E1 7.4415,E2 499.1619} C_DIS
LIN {X 87.8359,Y -109.0831,Z 175,A -48.6033,B 7.3281,C 0.3835,E1 7.4383,E2 500.6284} C_DIS
LIN {X 84.1905,Y -111.9208,Z 175,A -50.5619,B 7.3278,C 0.3882,E1 7.4339,E2 502.5977} C_DIS
LIN {X 78.2675,Y -116.1401,Z 175,A -53.1519,B 7.3279,C 0.3863,E1 7.4281,E2 505.1399} C_DIS
LIN {X 70.5725,Y -120.9703,Z 175,A -57.1001,B 7.3274,C 0.3966,E1 7.4187,E2 509.1217} C_DIS
LIN {X 66.6536,Y -123.1735,Z 175,A -58.9454,B 7.3272,C 0.3994,E1 7.4142,E2 510.9694} C_DIS
LIN {X 63.038,Y -125.0608,Z 175,A -60.4845,B 7.3272,C 0.3994,E1 7.4104,E2 512.4927} C_DIS
LIN {X 60.4092,Y -126.3504,Z 175,A -61.6212,B 7.3272,C 0.3999,E1 7.4075,E2 513.6224} C_DIS
LIN {X 54.3166,Y -129.0874,Z 175,A -64.1955,B 7.3272,C 0.4005,E1 7.401,E2 516.178} C_DIS
LIN {X 50.1233,Y -130.7739,Z 175,A -66.191,B 7.3269,C 0.4053,E1 7.3958,E2 518.1942} C_DIS
LIN {X 47.1871,Y -131.8606,Z 175,A -68.1099,B 7.3262,C 0.418,E1 7.3905,E2 520.1973} C_DIS
LIN {X 42.19,Y -133.5437,Z 175,A -69.5877,B 7.3267,C 0.4082,E1 7.3868,E2 521.588} C_DIS
LIN {X 38.6701,Y -134.6063,Z 175,A -71.1256,B 7.3267,C 0.4102,E1 7.3827,E2 523.1315} C_DIS
LIN {X 32.0393,Y -136.3374,Z 175,A -73.8873,B 7.3265,C 0.4118,E1 7.3752,E2 525.8896} C_DIS
LIN {X 29.1376,Y -136.9852,Z 175,A -75.2468,B 7.3263,C 0.4151,E1 7.3714,E2 527.2686} C_DIS
LIN {X 23.4806,Y -138.0675,Z 175,A -77.68,B 7.3262,C 0.418,E1 7.3647,E2 529.7134} C_DIS
LIN {X 17.3114,Y -138.9772,Z 175,A -79.9505,B 7.3264,C 0.4145,E1 7.3585,E2 531.9486} C_DIS
LIN {X 14.6083,Y -139.2859,Z 175,A -81.1938,B 7.3262,C 0.4172,E1 7.355,E2 533.2096} C_DIS
LIN {X 10.3905,Y -139.6635,Z 175,A -82.8856,B 7.3262,C 0.4171,E1 7.3503,E2 534.8969} C_DIS
LIN {X 6.2928,Y -139.9099,Z 175,A -84.6427,B 7.3262,C 0.4189,E1 7.3454,E2 536.6652} C_DIS
LIN {X 2.1044,Y -140.0338,Z 175,A -86.2134,B 7.3262,C 0.4168,E1 7.3411,E2 538.2178} C_DIS
LIN {X 2.1044,Y -140.0338,Z 175,A -86.2134,B 7.3262,C 0.4168,E1 7.3411,E2 538.2178} C_DIS
Enddeposition()
LIN {X 1.0389,Y -140.9505,Z 175,A -86.3019,B 7.3265,C 0.4152,E1 7.341,E2 538.2939} C_DIS
Startdeposition()
$VEL.CP = VEL_PRINT
LIN {X 3.6478,Y -140.909,Z 175,A -84.8844,B 7.3268,C 0.4089,E1 7.3451,E2 536.8283} C_DIS
LIN {X 8.0211,Y -140.729,Z 175,A -83.1109,B 7.3268,C 0.4085,E1 7.35,E2 535.0547} C_DIS
LIN {X 11.3908,Y -140.4956,Z 175,A -81.8153,B 7.3268,C 0.4094,E1 7.3536,E2 533.7687} C_DIS
LIN {X 14.4453,Y -140.2151,Z 175,A -80.6447,B 7.3268,C 0.4102,E1 7.3568,E2 532.6076} C_DIS
LIN {X 17.4694,Y -139.8712,Z 175,A -78.8705,B 7.3273,C 0.4002,E1 7.362,E2 530.7606} C_DIS
LIN {X 21.5869,Y -139.2929,Z 175,A -77.5754,B 7.327,C 0.4063,E1 7.3654,E2 529.5175} C_DIS
LIN {X 26.2146,Y -138.4968,Z 175,A -75.8313,B 7.3269,C 0.408,E1 7.3701,E2 527.7944} C_DIS
LIN {X 29.4301,Y -137.8494,Z 175,A -74.6126,B 7.3269,C 0.4091,E1 7.3734,E2 526.5901} C_DIS
LIN {X 32.7603,Y -137.096,Z 175,A -73.2411,B 7.3269,C 0.4083,E1 7.3772,E2 525.2199} C_DIS
LIN {X 35.808,Y -136.3325,Z 175,A -71.5665,B 7.3273,C 0.4001,E1 7.3818,E2 523.4913} C_DIS
LIN {X 40.7689,Y -134.9319,Z 175,A -69.6592,B 7.3273,C 0.4016,E1 7.3869,E2 521.6078} C_DIS
LIN {X 45.0981,Y -133.5476,Z 175,A -67.7602,B 7.3273,C 0.3988,E1 7.3919,E2 519.7005} C_DIS
LIN {X 49.0783,Y -132.136,Z 175,A -66.2687,B 7.3273,C 0.401,E1 7.3958,E2 518.2379} C_DIS
LIN {X 51.8542,Y -131.0736,Z 175,A -64.8164,B 7.3276,C 0.3952,E1 7.3997,E2 516.752} C_DIS
LIN {X 54.9836,Y -129.7912,Z 175,A -63.1489,B 7.3279,C 0.3881,E1 7.4041,E2 515.0442} C_DIS
LIN {X 58.7476,Y -128.1302,Z 175,A -61.8995,B 7.3276,C 0.3938,E1 7.4071,E2 513.8502} C_DIS
LIN {X 61.4854,Y -126.8408,Z 175,A -60.5286,B 7.3279,C 0.3895,E1 7.4106,E2 512.4596} C_DIS
LIN {X 64.9904,Y -125.0801,Z 175,A -59.0591,B 7.3279,C 0.3895,E1 7.4142,E2 511.0055} C_DIS
LIN {X 68.711,Y -123.077,Z 175,A -56.886,B 7.3284,C 0.3785,E1 7.4197,E2 508.7698} C_DIS
LIN {X 72.8353,Y -120.6815,Z 175,A -55.4482,B 7.3281,C 0.3848,E1 7.423,E2 507.3977} C_DIS
LIN {X 76.5798,Y -118.3409,Z 175,A -53.6335,B 7.3283,C 0.3815,E1 7.4272,E2 505.5789} C_DIS
LIN {X 79.149,Y -116.6381,Z 175,A -52.3143,B 7.3285,C 0.3782,E1 7.4303,E2 504.2497} C_DIS
LIN {X 83.1499,Y -113.821,Z 175,A -50.4646,B 7.3285,C 0.3773,E1 7.4345,E2 502.4169} C_DIS
LIN {X 86.4007,Y -111.3728,Z 175,A -48.8607,B 7.3286,C 0.3752,E1 7.438,E2 500.8182} C_DIS
LIN {X 89.4754,Y -108.9186,Z 175,A -47.2217,B 7.3288,C 0.3714,E1 7.4416,E2 499.1725} C_DIS
LIN {X 92.562,Y -106.3075,Z 175,A -45.6115,B 7.3289,C 0.3688,E1 7.445,E2 497.5651} C_DIS
LIN {X 95.7394,Y -103.4557,Z 175,A -43.9171,B 7.3291,C 0.3661,E1 7.4485,E2 495.8746} C_DIS
LIN {X 98.8118,Y -100.5247,Z 175,A -42.2536,B 7.3291,C 0.3637,E1 7.4518,E2 494.2179} C_DIS
LIN {X 101.6221,Y -97.6837,Z 175,A -40.7039,B 7.3293,C 0.3617,E1 7.4548,E2 492.6766} C_DIS
LIN {X 104.3547,Y -94.7579,Z 175,A -39.0325,B 7.3295,C 0.3573,E1 7.458,E2 490.9977} C_DIS
LIN {X 106.9981,Y -91.7631,Z 175,A -37.4553,B 7.3296,C 0.3546,E1 7.4609,E2 489.4252} C_DIS
LIN {X 109.4619,Y -88.8102,Z 175,A -36.0199,B 7.3296,C 0.3535,E1 7.4634,E2 488.0053} C_DIS
LIN {X 111.6289,Y -86.0696,Z 175,A -34.1362,B 7.3303,C 0.3411,E1 7.4667,E2 486.0583} C_DIS
LIN {X 114.0628,Y -82.8171,Z 175,A -32.7821,B 7.3302,C 0.343,E1 7.4689,E2 484.7424} C_DIS
LIN {X 116.8332,Y -78.8608,Z 175,A -30.9101,B 7.3303,C 0.34,E1 7.4718,E2 482.8806} C_DIS
LIN {X 120.6079,Y -72.957,Z 175,A -28.132,B 7.3306,C 0.3344,E1 7.4759,E2 480.1091} C_DIS
LIN {X 122.7863,Y -69.2283,Z 175,A -26.3574,B 7.3308,C 0.3295,E1 7.4784,E2 478.3303} C_DIS
LIN {X 124.7914,Y -65.5401,Z 175,A -24.2345,B 7.3313,C 0.3168,E1 7.4813,E2 476.15} C_DIS
LIN {X 127.004,Y -61.1438,Z 175,A -22.8436,B 7.3311,C 0.3237,E1 7.4829,E2 474.8385} C_DIS
LIN {X 128.7488,Y -57.3776,Z 175,A -21.2129,B 7.3311,C 0.3203,E1 7.4847,E2 473.2137} C_DIS
LIN {X 129.8283,Y -54.8946,Z 175,A -20.1721,B 7.3313,C 0.3186,E1 7.4859,E2 472.1798} C_DIS
LIN {X 131.1716,Y -51.6021,Z 175,A -18.7717,B 7.3314,C 0.3156,E1 7.4873,E2 470.7839} C_DIS
LIN {X 132.1558,Y -49.0252,Z 175,A -17.4482,B 7.3317,C 0.3085,E1 7.4887,E2 469.4326} C_DIS
LIN {X 133.4334,Y -45.4378,Z 175,A -16.0522,B 7.3317,C 0.3073,E1 7.4899,E2 468.0552} C_DIS
LIN {X 134.4694,Y -42.2714,Z 175,A -13.9747,B 7.3325,C 0.2891,E1 7.4917,E2 465.8801} C_DIS
LIN {X 136.1222,Y -36.5963,Z 175,A -12.3042,B 7.3322,C 0.297,E1 7.4929,E2 464.3049} C_DIS
LIN {X 137.026,Y -33.0507,Z 175,A -10.9646,B 7.3322,C 0.2958,E1 7.4938,E2 462.9834} C_DIS
LIN {X 137.8709,Y -29.3308,Z 175,A -9.1616,B 7.3326,C 0.2863,E1 7.4949,E2 461.1456} C_DIS
LIN {X 138.6679,Y -25.2969,Z 175,A -7.7649,B 7.3326,C 0.2871,E1 7.4956,E2 459.7837} C_DIS
LIN {X 139.1784,Y -22.3266,Z 175,A -6.393,B 7.3328,C 0.2807,E1 7.4962,E2 458.3914} C_DIS
LIN {X 139.8534,Y -17.6084,Z 175,A -4.6341,B 7.3328,C 0.2787,E1 7.4969,E2 456.6542} C_DIS
LIN {X 140.2111,Y -14.4826,Z 175,A -3.4095,B 7.333,C 0.2761,E1 7.4972,E2 455.4356} C_DIS
LIN {X 140.5964,Y -10.0627,Z 175,A -1.5377,B 7.3332,C 0.2695,E1 7.4976,E2 453.5532} C_DIS
LIN {X 140.8371,Y -5.7953,Z 175,A 0.1114,B 7.3333,C 0.2663,E1 7.4979,E2 451.9141} C_DIS
LIN {X 140.9474,Y -1.6798,Z 175,A 1.6406,B 7.3334,C 0.2644,E1 7.4979,E2 450.4025} C_DIS
LIN {X 140.9498,Y 1.5075,Z 175,A 3.1185,B 7.3337,C 0.257,E1 7.4979,E2 448.8995} C_DIS
LIN {X 140.8557,Y 5.3168,Z 175,A 4.38,B 7.3337,C 0.2582,E1 7.4979,E2 447.6744} C_DIS
LIN {X 140.7357,Y 7.9113,Z 175,A 5.6773,B 7.3339,C 0.2504,E1 7.4976,E2 446.3446} C_DIS
LIN {X 140.4225,Y 12.256,Z 175,A 7.4165,B 7.3341,C 0.246,E1 7.4972,E2 444.608} C_DIS
LIN {X 140.0085,Y 16.3185,Z 175,A 9.0381,B 7.3341,C 0.242,E1 7.4967,E2 442.9901} C_DIS
LIN {X 139.3734,Y 21.0672,Z 175,A 10.724,B 7.3341,C 0.2416,E1 7.4961,E2 441.337} C_DIS
LIN {X 138.7925,Y 24.6008,Z 175,A 12.151,B 7.3343,C 0.2381,E1 7.4954,E2 439.9127} C_DIS
LIN {X 138.1368,Y 28.0486,Z 175,A 13.5158,B 7.3344,C 0.2353,E1 7.4947,E2 438.5548} C_DIS
LIN {X 137.596,Y 30.6021,Z 175,A 14.8482,B 7.3347,C 0.227,E1 7.4939,E2 437.1862} C_DIS
LIN {X 136.7467,Y 34.1916,Z 175,A 16.2632,B 7.3347,C 0.2244,E1 7.493,E2 435.7811} C_DIS
LIN {X 135.802,Y 37.7668,Z 175,A 17.6421,B 7.3347,C 0.2227,E1 7.492,E2 434.4175} C_DIS
LIN {X 134.7974,Y 41.2082,Z 175,A 19.1124,B 7.3349,C 0.2185,E1 7.4908,E2 432.9444} C_DIS
LIN {X 133.7008,Y 44.6382,Z 175,A 20.4043,B 7.3349,C 0.2179,E1 7.4897,E2 431.6739} C_DIS
LIN {X 132.6956,Y 47.5436,Z 175,A 21.7526,B 7.3351,C 0.2126,E1 7.4884,E2 430.312} C_DIS
LIN {X 131.205,Y 51.5161,Z 175,A 23.2886,B 7.3351,C 0.2116,E1 7.4869,E2 428.7994} C_DIS
LIN {X 129.8257,Y 54.9008,Z 175,A 25.0118,B 7.3354,C 0.2031,E1 7.485,E2 427.0445} C_DIS
LIN {X 128.0362,Y 58.9508,Z 175,A 26.6772,B 7.3354,C 0.201,E1 7.4831,E2 425.3955} C_DIS
LIN {X 126.1039,Y 62.9817,Z 175,A 28.5368,B 7.3356,C 0.1955,E1 7.4808,E2 423.5293} C_DIS
LIN {X 123.9863,Y 67.0563,Z 175,A 30.2622,B 7.3356,C 0.1935,E1 7.4786,E2 421.8214} C_DIS
LIN {X 121.9648,Y 70.6652,Z 175,A 31.9652,B 7.3357,C 0.1889,E1 7.4763,E2 420.1147} C_DIS
LIN {X 119.8975,Y 74.1198,Z 175,A 33.6695,B 7.3359,C 0.1836,E1 7.4738,E2 418.4008} C_DIS
LIN {X 117.4985,Y 77.867,Z 175,A 35.3189,B 7.3359,C 0.1823,E1 7.4713,E2 416.7712} C_DIS
LIN {X 115.399,Y 80.9456,Z 175,A 36.9173,B 7.336,C 0.1772,E1 7.4687,E2 415.1612} C_DIS
LIN {X 112.7179,Y 84.639,Z 175,A 38.4432,B 7.336,C 0.1792,E1 7.4663,E2 413.6771} C_DIS
LIN {X 107.8858,Y 90.7175,Z 175,A 41.8493,B 7.3363,C 0.1674,E1 7.4603,E2 410.2378} C_DIS
LIN {X 104.9759,Y 94.0693,Z 175,A 43.5652,B 7.3363,C 0.1652,E1 7.4571,E2 408.5327} C_DIS
LIN {X 102.2397,Y 97.0372,Z 175,A 45.1799,B 7.3363,C 0.1623,E1 7.454,E2 406.921} C_DIS
LIN {X 99.1977,Y 100.1441,Z 175,A 46.8152,B 7.3363,C 0.1612,E1 7.4508,E2 405.3022} C_DIS
LIN {X 93.2603,Y 105.6954,Z 175,A 50.2229,B 7.3366,C 0.1529,E1 7.4438,E2 401.8805} C_DIS
LIN {X 89.9836,Y 108.4986,Z 175,A 51.9593,B 7.3366,C 0.1499,E1 7.4401,E2 400.1458} C_DIS
LIN {X 86.372,Y 111.3951,Z 175,A 53.8197,B 7.3366,C 0.147,E1 7.436,E2 398.2879} C_DIS
LIN {X 82.6473,Y 114.1859,Z 175,A 55.6688,B 7.3367,C 0.1445,E1 7.4319,E2 396.4441} C_DIS
LIN {X 78.6829,Y 116.9536,Z 175,A 57.5847,B 7.3367,C 0.1423,E1 7.4275,E2 394.5344} C_DIS
LIN {X 75.4157,Y 119.0861,Z 175,A 59.1505,B 7.3368,C 0.1402,E1 7.4238,E2 392.971} C_DIS
LIN {X 71.7958,Y 121.3035,Z 175,A 60.944,B 7.3368,C 0.1364,E1 7.4195,E2 391.1687} C_DIS
LIN {X 67.747,Y 123.6099,Z 175,A 62.5948,B 7.3368,C 0.1381,E1 7.4156,E2 389.549} C_DIS
LIN {X 63.2567,Y 125.9667,Z 175,A 64.7486,B 7.3369,C 0.1337,E1 7.4102,E2 387.3835} C_DIS
LIN {X 59.5443,Y 127.7618,Z 175,A 66.354,B 7.3369,C 0.1329,E1 7.4062,E2 385.7872} C_DIS
LIN {X 56.1797,Y 129.2762,Z 175,A 67.6755,B 7.3369,C 0.1343,E1 7.4028,E2 384.4885} C_DIS
LIN {X 53.2358,Y 130.5171,Z 175,A 69.0736,B 7.3369,C 0.1311,E1 7.3992,E2 383.0779} C_DIS
LIN {X 49.8541,Y 131.8454,Z 175,A 70.5062,B 7.337,C 0.1304,E1 7.3955,E2 381.6511} C_DIS
LIN {X 46.8727,Y 132.9359,Z 175,A 72.0352,B 7.337,C 0.125,E1 7.3914,E2 380.0918} C_DIS
LIN {X 42.5417,Y 134.383,Z 175,A 73.7556,B 7.337,C 0.1257,E1 7.3869,E2 378.389} C_DIS
LIN {X 38.7437,Y 135.5288,Z 175,A 75.4834,B 7.3371,C 0.1224,E1 7.3822,E2 376.6468} C_DIS
LIN {X 35.4559,Y 136.4258,Z 175,A 77.0457,B 7.3372,C 0.1183,E1 7.3779,E2 375.0622} C_DIS
LIN {X 32.1695,Y 137.2379,Z 175,A 78.0961,B 7.3372,C 0.123,E1 7.3752,E2 374.0538} C_DIS
LIN {X 28.6663,Y 138.0111,Z 175,A 79.6954,B 7.3372,C 0.1197,E1 7.3708,E2 372.4368} C_DIS
LIN {X 25.0639,Y 138.7096,Z 175,A 80.8969,B 7.3372,C 0.1238,E1 7.3676,E2 371.2728} C_DIS
LIN {X 21.8729,Y 139.2487,Z 175,A 82.3987,B 7.3372,C 0.1201,E1 7.3634,E2 369.7477} C_DIS
LIN {X 18.6614,Y 139.7154,Z 175,A 83.6092,B 7.3372,C 0.1214,E1 7.3601,E2 368.5514} C_DIS
LIN {X 15.8267,Y 140.0665,Z 175,A 84.8012,B 7.3372,C 0.1205,E1 7.3567,E2 367.3559} C_DIS
LIN {X 12.9813,Y 140.3577,Z 175,A 85.975,B 7.3372,C 0.1199,E1 7.3535,E2 366.1811} C_DIS
LIN {X 10.0811,Y 140.595,Z 175,A 87.1911,B 7.3372,C 0.1191,E1 7.3501,E2 364.9612} C_DIS
LIN {X 5.8852,Y 140.8336,Z 175,A 88.7619,B 7.3372,C 0.1211,E1 7.3457,E2 363.4086} C_DIS
LIN {X 3.3813,Y 140.9164,Z 175,A 89.8701,B 7.3372,C 0.1196,E1 7.3426,E2 362.2894} C_DIS
LIN {X 0.3339,Y 140.9563,Z 175,A 91.2692,B 7.3372,C 0.1169,E1 7.3387,E2 360.8704} C_DIS
LIN {X -3.8296,Y 140.9039,Z 175,A 92.9163,B 7.3372,C 0.1178,E1 7.3341,E2 359.2298} C_DIS
LIN {X -7.9191,Y 140.7352,Z 175,A 94.4639,B 7.3372,C 0.1199,E1 7.3298,E2 357.698} C_DIS
LIN {X -10.4439,Y 140.5685,Z 175,A 95.5574,B 7.3372,C 0.119,E1 7.3267,E2 356.5967} C_DIS
LIN {X -13.9773,Y 140.262,Z 175,A 96.9593,B 7.3372,C 0.1201,E1 7.3228,E2 355.2006} C_DIS
LIN {X -17.8947,Y 139.8159,Z 175,A 98.6162,B 7.3372,C 0.1197,E1 7.3182,E2 353.5377} C_DIS
LIN {X -22.6513,Y 139.1246,Z 175,A 100.935,B 7.3372,C 0.1148,E1 7.3117,E2 351.1733} C_DIS
LIN {X -26.415,Y 138.4585,Z 175,A 102.8212,B 7.3373,C 0.1104,E1 7.3064,E2 349.2453} C_DIS
LIN {X -32.0557,Y 137.2639,Z 175,A 104.4162,B 7.3371,C 0.1236,E1 7.3024,E2 347.7478} C_DIS
LIN {X -37.1191,Y 135.9828,Z 175,A 106.7423,B 7.3371,C 0.122,E1 7.296,E2 345.3972} C_DIS
LIN {X -41.3202,Y 134.7631,Z 175,A 108.3928,B 7.3371,C 0.1254,E1 7.2916,E2 343.7641} C_DIS
LIN {X -44.6873,Y 133.6844,Z 175,A 109.692,B 7.3371,C 0.1288,E1 7.2882,E2 342.4834} C_DIS
LIN {X -47.8871,Y 132.5718,Z 175,A 111.3641,B 7.3371,C 0.1257,E1 7.2837,E2 340.7747} C_DIS
LIN {X -52.422,Y 130.8452,Z 175,A 113.222,B 7.3371,C 0.1295,E1 7.2789,E2 338.9329} C_DIS
LIN {X -55.8086,Y 129.4366,Z 175,A 114.722,B 7.337,C 0.131,E1 7.2751,E2 337.4328} C_DIS
LIN {X -58.7748,Y 128.1176,Z 175,A 116.308,B 7.337,C 0.1286,E1 7.271,E2 335.8139} C_DIS
LIN {X -61.768,Y 126.7026,Z 175,A 117.4821,B 7.337,C 0.1328,E1 7.2681,E2 334.6628} C_DIS
LIN {X -65.1417,Y 125.0006,Z 175,A 118.9843,B 7.337,C 0.1354,E1 7.2644,E2 333.1661} C_DIS
LIN {X -68.601,Y 123.1382,Z 175,A 120.7059,B 7.337,C 0.1357,E1 7.2601,E2 331.4299} C_DIS
LIN {X -72.4238,Y 120.9291,Z 175,A 122.3873,B 7.3368,C 0.14,E1 7.2561,E2 329.7644} C_DIS
LIN {X -75.9409,Y 118.7517,Z 175,A 124.0826,B 7.3368,C 0.1424,E1 7.2521,E2 328.0688} C_DIS
LIN {X -79.0996,Y 116.6715,Z 175,A 125.6487,B 7.3368,C 0.1445,E1 7.2484,E2 326.5003} C_DIS
LIN {X -81.2528,Y 115.1823,Z 175,A 127.2482,B 7.3368,C 0.1384,E1 7.2447,E2 324.8331} C_DIS
LIN {X -85.0907,Y 112.377,Z 175,A 129.4186,B 7.3368,C 0.1384,E1 7.2398,E2 322.6338} C_DIS
LIN {X -89.7324,Y 108.7066,Z 175,A 130.9999,B 7.3365,C 0.1546,E1 7.2366,E2 321.1604} C_DIS
LIN {X -94.3089,Y 104.7611,Z 175,A 133.7152,B 7.3365,C 0.1556,E1 7.2308,E2 318.4143} C_DIS
LIN {X -97.5557,Y 101.7444,Z 175,A 135.4741,B 7.3365,C 0.1598,E1 7.2272,E2 316.6625} C_DIS
LIN {X -101.0604,Y 98.2643,Z 175,A 138.1513,B 7.3365,C 0.1544,E1 7.2219,E2 313.901} C_DIS
LIN {X -104.8779,Y 94.1788,Z 175,A 139.6494,B 7.3362,C 0.1702,E1 7.2192,E2 312.5047} C_DIS
LIN {X -107.0361,Y 91.7186,Z 175,A 141.5183,B 7.3362,C 0.1656,E1 7.2157,E2 310.568} C_DIS
LIN {X -109.5996,Y 88.6394,Z 175,A 142.6929,B 7.3361,C 0.1756,E1 7.2137,E2 309.4532} C_DIS
LIN {X -112.6526,Y 84.7255,Z 175,A 144.8419,B 7.336,C 0.1784,E1 7.21,E2 307.2894} C_DIS
LIN {X -115.0456,Y 81.4466,Z 175,A 146.5539,B 7.336,C 0.1814,E1 7.2072,E2 305.571} C_DIS
LIN {X -117.3417,Y 78.1021,Z 175,A 148.1182,B 7.3358,C 0.1865,E1 7.2048,E2 304.0192} C_DIS
LIN {X -120.1005,Y 73.7893,Z 175,A 150.3823,B 7.3358,C 0.1891,E1 7.2014,E2 301.7335} C_DIS
LIN {X -122.0509,Y 70.5165,Z 175,A 151.9411,B 7.3356,C 0.1928,E1 7.1992,E2 300.175} C_DIS
LIN {X -124.3346,Y 66.4079,Z 175,A 153.9554,B 7.3356,C 0.1962,E1 7.1965,E2 298.1492} C_DIS
LIN {X -126.2608,Y 62.6638,Z 175,A 155.3479,B 7.3353,C 0.205,E1 7.1948,E2 296.7992} C_DIS
LIN {X -128.9742,Y 56.8737,Z 175,A 158.3138,B 7.3353,C 0.2069,E1 7.1913,E2 293.789} C_DIS
LIN {X -130.6016,Y 53.0262,Z 175,A 159.831,B 7.3351,C 0.2138,E1 7.1897,E2 292.2966} C_DIS
LIN {X -131.9213,Y 49.6515,Z 175,A 161.4356,B 7.335,C 0.216,E1 7.1881,E2 290.6765} C_DIS
LIN {X -133.107,Y 46.3792,Z 175,A 162.6985,B 7.3348,C 0.2219,E1 7.1869,E2 289.4344} C_DIS
LIN {X -133.9659,Y 43.842,Z 175,A 163.9685,B 7.3348,C 0.2225,E1 7.1857,E2 288.1422} C_DIS
LIN {X -135.1471,Y 40.0491,Z 175,A 165.6328,B 7.3347,C 0.2263,E1 7.1844,E2 286.4731} C_DIS
LIN {X -136.0304,Y 36.9406,Z 175,A 166.8765,B 7.3345,C 0.2309,E1 7.1835,E2 285.2397} C_DIS
LIN {X -136.9548,Y 33.3463,Z 175,A 168.387,B 7.3345,C 0.2351,E1 7.1824,E2 283.7303} C_DIS
LIN {X -137.685,Y 30.1918,Z 175,A 169.6883,B 7.3343,C 0.239,E1 7.1816,E2 282.4322} C_DIS
LIN {X -138.8216,Y 24.4383,Z 175,A 172.1838,B 7.3341,C 0.2442,E1 7.1803,E2 279.9246} C_DIS
LIN {X -139.8772,Y 17.4197,Z 175,A 175.8436,B 7.3341,C 0.242,E1 7.1789,E2 276.1669} C_DIS
LIN {X -140.4145,Y 12.3512,Z 175,A 177.5347,B 7.3338,C 0.2531,E1 7.1785,E2 274.5273} C_DIS
LIN {X -140.7753,Y 7.1341,Z 175,A 179.4975,B 7.3335,C 0.2614,E1 7.1781,E2 272.5875} C_DIS
LIN {X -140.9195,Y 3.2676,Z 175,A -178.9687,B 7.3333,C 0.2665,E1 7.178,E2 271.0602} C_DIS
LIN {X -140.9511,Y -1.3264,Z 175,A -176.7197,B 7.3333,C 0.2667,E1 7.178,E2 268.7633} C_DIS
LIN {X -140.8844,Y -4.5326,Z 175,A -175.5205,B 7.3331,C 0.2719,E1 7.1781,E2 267.5787} C_DIS
LIN {X -140.6996,Y -8.4974,Z 175,A -173.963,B 7.3329,C 0.2772,E1 7.1783,E2 266.0297} C_DIS
LIN {X -140.2689,Y -13.9055,Z 175,A -171.4485,B 7.3329,C 0.2794,E1 7.179,E2 263.4768} C_DIS
LIN {X -139.8748,Y -17.4394,Z 175,A -169.661,B 7.3329,C 0.2788,E1 7.1796,E2 261.6456} C_DIS
LIN {X -139.1461,Y -22.5243,Z 175,A -168.0855,B 7.3324,C 0.2917,E1 7.1803,E2 260.1389} C_DIS
LIN {X -138.4864,Y -26.2692,Z 175,A -166.5689,B 7.3322,C 0.2964,E1 7.181,E2 258.6272} C_DIS
LIN {X -137.8519,Y -29.4185,Z 175,A -165.3193,B 7.332,C 0.3009,E1 7.1817,E2 257.3859} C_DIS
LIN {X -137.1097,Y -32.7036,Z 175,A -163.9401,B 7.3319,C 0.3045,E1 7.1826,E2 256.0063} C_DIS
LIN {X -136.3237,Y -35.841,Z 175,A -162.55,B 7.3318,C 0.3072,E1 7.1836,E2 254.6074} C_DIS
LIN {X -135.3211,Y -39.4548,Z 175,A -160.997,B 7.3316,C 0.311,E1 7.1848,E2 253.0517} C_DIS
LIN {X -134.2649,Y -42.9114,Z 175,A -159.5057,B 7.3314,C 0.3146,E1 7.186,E2 251.5585} C_DIS
LIN {X -133.303,Y -45.8136,Z 175,A -158.3764,B 7.3312,C 0.3196,E1 7.187,E2 250.4449} C_DIS
LIN {X -132.3271,Y -48.5658,Z 175,A -156.8851,B 7.3312,C 0.3186,E1 7.1885,E2 248.9146} C_DIS
LIN {X -130.7957,Y -52.5447,Z 175,A -155.2747,B 7.331,C 0.3248,E1 7.1901,E2 247.3213} C_DIS
LIN {X -129.5044,Y -55.652,Z 175,A -153.801,B 7.331,C 0.3269,E1 7.1917,E2 245.8345} C_DIS
LIN {X -128.1628,Y -58.6771,Z 175,A -152.4311,B 7.3308,C 0.3301,E1 7.1933,E2 244.4623} C_DIS
LIN {X -126.5202,Y -62.1378,Z 175,A -150.9377,B 7.3305,C 0.3349,E1 7.1951,E2 242.9781} C_DIS
LIN {X -124.8139,Y -65.4974,Z 175,A -148.5118,B 7.3309,C 0.3262,E1 7.1984,E2 240.435} C_DIS
LIN {X -121.7945,Y -70.9594,Z 175,A -146.6207,B 7.3302,C 0.3416,E1 7.2009,E2 238.6308} C_DIS
LIN {X -119.4317,Y -74.8682,Z 175,A -144.6231,B 7.3302,C 0.344,E1 7.2038,E2 236.6155} C_DIS
LIN {X -116.549,Y -79.2806,Z 175,A -142.5665,B 7.3298,C 0.3503,E1 7.207,E2 234.5713} C_DIS
LIN {X -113.9193,Y -83.015,Z 175,A -140.6653,B 7.3297,C 0.3539,E1 7.2101,E2 232.665} C_DIS
LIN {X -111.1491,Y -86.6893,Z 175,A -138.7612,B 7.3295,C 0.3575,E1 7.2134,E2 230.7571} C_DIS
LIN {X -108.3175,Y -90.2023,Z 175,A -136.9951,B 7.3292,C 0.3625,E1 7.2165,E2 229.0008} C_DIS
LIN {X -104.945,Y -94.1039,Z 175,A -134.8105,B 7.3291,C 0.3656,E1 7.2205,E2 226.8051} C_DIS
LIN {X -101.8026,Y -97.4948,Z 175,A -132.9428,B 7.3289,C 0.3696,E1 7.2241,E2 224.9396} C_DIS
LIN {X -98.9038,Y -100.4345,Z 175,A -131.4353,B 7.3286,C 0.3754,E1 7.227,E2 223.4551} C_DIS
LIN {X -96.2334,Y -102.9959,Z 175,A -129.6528,B 7.3286,C 0.3741,E1 7.2307,E2 221.6362} C_DIS
LIN {X -92.8537,Y -106.0529,Z 175,A -127.8118,B 7.3285,C 0.3777,E1 7.2345,E2 219.7971} C_DIS
LIN {X -89.5761,Y -108.836,Z 175,A -126.0034,B 7.3284,C 0.3799,E1 7.2384,E2 217.981} C_DIS
LIN {X -86.01,Y -111.6756,Z 175,A -124.1248,B 7.3282,C 0.3826,E1 7.2426,E2 216.0993} C_DIS
LIN {X -83.607,Y -113.4852,Z 175,A -122.8864,B 7.3282,C 0.3844,E1 7.2454,E2 214.859} C_DIS
LIN {X -79.6703,Y -116.2826,Z 175,A -120.9358,B 7.328,C 0.3876,E1 7.2498,E2 212.9102} C_DIS
LIN {X -75.849,Y -118.8105,Z 175,A -119.0611,B 7.3278,C 0.3902,E1 7.2542,E2 211.034} C_DIS
LIN {X -71.92,Y -121.2294,Z 175,A -117.1244,B 7.3278,C 0.3918,E1 7.2589,E2 209.0893} C_DIS
LIN {X -69.1684,Y -122.8199,Z 175,A -115.4757,B 7.3279,C 0.388,E1 7.263,E2 207.3931} C_DIS
LIN {X -65.5236,Y -124.8001,Z 175,A -114.267,B 7.3274,C 0.3975,E1 7.2658,E2 206.248} C_DIS
LIN {X -62.7275,Y -126.2293,Z 175,A -112.9087,B 7.3274,C 0.3978,E1 7.2692,E2 204.8788} C_DIS
LIN {X -59.3268,Y -127.8624,Z 175,A -111.2046,B 7.3274,C 0.3968,E1 7.2736,E2 203.1518} C_DIS
LIN {X -55.056,Y -129.7609,Z 175,A -109.491,B 7.3272,C 0.4017,E1 7.2779,E2 201.463} C_DIS
LIN {X -51.5904,Y -131.1761,Z 175,A -108.0721,B 7.327,C 0.4048,E1 7.2816,E2 200.0575} C_DIS
LIN {X -48.0902,Y -132.4985,Z 175,A -106.4061,B 7.327,C 0.4039,E1 7.286,E2 198.372} C_DIS
LIN {X -44.4384,Y -133.7673,Z 175,A -104.8615,B 7.327,C 0.4056,E1 7.29,E2 196.8306} C_DIS
LIN {X -41.4644,Y -134.719,Z 175,A -103.5677,B 7.327,C 0.4061,E1 7.2935,E2 195.5334} C_DIS
LIN {X -37.0551,Y -135.9999,Z 175,A -101.5641,B 7.327,C 0.4051,E1 7.2989,E2 193.5112} C_DIS
LIN {X -33.5006,Y -136.9176,Z 175,A -100.0396,B 7.327,C 0.4055,E1 7.3031,E2 191.982} C_DIS
LIN {X -28.6408,Y -138.0163,Z 175,A -98.2834,B 7.3267,C 0.4109,E1 7.3078,E2 190.2611} C_DIS
LIN {X -25.5935,Y -138.6149,Z 175,A -96.6456,B 7.327,C 0.4052,E1 7.3124,E2 188.5728} C_DIS
LIN {X -20.8712,Y -139.4038,Z 175,A -94.8031,B 7.3269,C 0.4076,E1 7.3175,E2 186.7435} C_DIS
LIN {X -16.5476,Y -139.9812,Z 175,A -93.1146,B 7.3268,C 0.4094,E1 7.3221,E2 185.0657} C_DIS
LIN {X -12.0554,Y -140.4395,Z 175,A -91.3033,B 7.3268,C 0.4101,E1 7.3271,E2 183.2569} C_DIS
LIN {X -8.4007,Y -140.7056,Z 175,A -89.7401,B 7.3268,C 0.4089,E1 7.3315,E2 181.6832} C_DIS
LIN {X -4.1477,Y -140.8951,Z 175,A -88.1813,B 7.3267,C 0.4118,E1 7.3358,E2 180.1466} C_DIS
LIN {X -1.0393,Y -140.9524,Z 175,A -86.984,B 7.3266,C 0.4129,E1 7.3391,E2 178.9576} C_DIS
LIN {X 1.0389,Y -140.9505,Z 175,A -86.2994,B 7.3264,C 0.4155,E1 7.341,E2 178.2938} C_DIS
Enddeposition()
LIN {X 1.0389,Y -140.9505,Z 175,A -86.2994,B 7.3264,C 0.4155,E1 7.341,E2 178.2938} C_DIS
Startdeposition()
$VEL.CP = VEL_PRINT
LIN {X 0.0011,Y -141.8646,Z 175,A -87.1107,B 7.3257,C 0.4265,E1 7.3384,E2 179.1912} C_DIS
LIN {X -4.3114,Y -141.7974,Z 175,A -88.8742,B 7.3257,C 0.427,E1 7.3335,E2 180.9582} C_DIS
LIN {X -8.4267,Y -141.6122,Z 175,A -90.4337,B 7.3258,C 0.4251,E1 7.3292,E2 182.5045} C_DIS
LIN {X -11.9101,Y -141.3615,Z 175,A -91.8752,B 7.3258,C 0.4255,E1 7.3251,E2 183.9507} C_DIS
LIN {X -15.6334,Y -140.999,Z 175,A -93.3411,B 7.3258,C 0.4245,E1 7.3211,E2 185.4112} C_DIS
LIN {X -19.0857,Y -140.5741,Z 175,A -94.7463,B 7.3258,C 0.4242,E1 7.3172,E2 186.817} C_DIS
LIN {X -22.5277,Y -140.0645,Z 175,A -96.1509,B 7.3258,C 0.4237,E1 7.3133,E2 188.2219} C_DIS
LIN {X -25.7094,Y -139.515,Z 175,A -97.535,B 7.3258,C 0.4245,E1 7.3095,E2 189.6172} C_DIS
LIN {X -29.3776,Y -138.7881,Z 175,A -98.9078,B 7.326,C 0.4216,E1 7.3058,E2 190.972} C_DIS
LIN {X -32.5158,Y -138.0874,Z 175,A -100.3408,B 7.326,C 0.4231,E1 7.3018,E2 192.4233} C_DIS
LIN {X -36.1479,Y -137.18,Z 175,A -101.8126,B 7.326,C 0.4215,E1 7.2978,E2 193.89} C_DIS
LIN {X -39.2445,Y -136.3273,Z 175,A -103.0342,B 7.3261,C 0.4194,E1 7.2946,E2 195.1019} C_DIS
LIN {X -42.5951,Y -135.3176,Z 175,A -104.6055,B 7.3261,C 0.4209,E1 7.2903,E2 196.6945} C_DIS
LIN {X -46.1506,Y -134.1457,Z 175,A -105.978,B 7.3262,C 0.4175,E1 7.2867,E2 198.0486} C_DIS
LIN {X -49.426,Y -132.9737,Z 175,A -107.4688,B 7.3262,C 0.4176,E1 7.2828,E2 199.551} C_DIS
LIN {X -52.4286,Y -131.8199,Z 175,A -108.7004,B 7.3264,C 0.4153,E1 7.2796,E2 200.774} C_DIS
LIN {X -55.6494,Y -130.4931,Z 175,A -110.1893,B 7.3264,C 0.4153,E1 7.2757,E2 202.2739} C_DIS
LIN {X -58.1576,Y -129.393,Z 175,A -111.312,B 7.3264,C 0.4143,E1 7.2729,E2 203.3987} C_DIS
LIN {X -61.4358,Y -127.8692,Z 175,A -112.7825,B 7.3265,C 0.4128,E1 7.2692,E2 204.8708} C_DIS
LIN {X -64.6618,Y -126.2685,Z 175,A -114.3056,B 7.3265,C 0.4122,E1 7.2653,E2 206.403} C_DIS
LIN {X -68.386,Y -124.2934,Z 175,A -116.0573,B 7.3266,C 0.4108,E1 7.261,E2 208.1613} C_DIS
LIN {X -72.0688,Y -122.1945,Z 175,A -117.7129,B 7.3268,C 0.4076,E1 7.257,E2 209.8093} C_DIS
LIN {X -75.549,Y -120.0739,Z 175,A -119.451,B 7.3268,C 0.4067,E1 7.2529,E2 211.5595} C_DIS
LIN {X -79.5355,Y -117.4711,Z 175,A -121.4242,B 7.327,C 0.4046,E1 7.2483,E2 213.5392} C_DIS
LIN {X -83.2016,Y -114.9037,Z 175,A -123.2545,B 7.3271,C 0.402,E1 7.2441,E2 215.3723} C_DIS
LIN {X -87.1486,Y -111.94,Z 175,A -125.1671,B 7.3274,C 0.3975,E1 7.2399,E2 217.2739} C_DIS
LIN {X -90.0974,Y -109.5809,Z 175,A -126.8091,B 7.3274,C 0.3966,E1 7.2363,E2 218.931} C_DIS
LIN {X -93.314,Y -106.8543,Z 175,A -128.4842,B 7.3276,C 0.3932,E1 7.2327,E2 220.6021} C_DIS
LIN {X -96.6504,Y -103.8463,Z 175,A -130.3458,B 7.3277,C 0.3905,E1 7.2289,E2 222.4695} C_DIS
LIN {X -99.795,Y -100.8285,Z 175,A -132.1431,B 7.3279,C 0.3876,E1 7.2253,E2 224.2712} C_DIS
LIN {X -102.8132,Y -97.7493,Z 175,A -133.7718,B 7.3281,C 0.3825,E1 7.2222,E2 225.8846} C_DIS
LIN {X -105.1059,Y -95.2791,Z 175,A -135.3099,B 7.3281,C 0.3823,E1 7.2192,E2 227.4454} C_DIS
LIN {X -107.9731,Y -92.0173,Z 175,A -136.9605,B 7.3284,C 0.3771,E1 7.2162,E2 229.0819} C_DIS
LIN {X -110.6799,Y -88.7439,Z 175,A -138.708,B 7.3286,C 0.3738,E1 7.2131,E2 230.8329} C_DIS
LIN {X -112.9826,Y -85.7932,Z 175,A -140.3798,B 7.3286,C 0.3728,E1 7.2103,E2 232.5252} C_DIS
LIN {X -115.9093,Y -81.7948,Z 175,A -142.2938,B 7.3289,C 0.367,E1 7.2072,E2 234.4269} C_DIS
LIN {X -118.362,Y -78.2038,Z 175,A -144.0847,B 7.3291,C 0.3634,E1 7.2044,E2 236.2214} C_DIS
LIN {X -120.7074,Y -74.5335,Z 175,A -145.9016,B 7.3293,C 0.36,E1 7.2016,E2 238.0451} C_DIS
LIN {X -122.9288,Y -70.8094,Z 175,A -147.6443,B 7.3295,C 0.3556,E1 7.1992,E2 239.7858} C_DIS
LIN {X -125.0366,Y -67.0167,Z 175,A -149.4495,B 7.3297,C 0.352,E1 7.1967,E2 241.5969} C_DIS
LIN {X -126.6559,Y -63.9009,Z 175,A -150.8569,B 7.3298,C 0.3483,E1 7.195,E2 243.0021} C_DIS
LIN {X -128.1844,Y -60.776,Z 175,A -152.2982,B 7.33,C 0.3452,E1 7.1932,E2 244.4473} C_DIS
LIN {X -129.6897,Y -57.4943,Z 175,A -153.7465,B 7.3302,C 0.3413,E1 7.1915,E2 245.8935} C_DIS
LIN {X -131.0679,Y -54.2788,Z 175,A -155.2082,B 7.3303,C 0.3382,E1 7.1899,E2 247.3607} C_DIS
LIN {X -132.6437,Y -50.307,Z 175,A -157.1121,B 7.3304,C 0.3361,E1 7.188,E2 249.2867} C_DIS
LIN {X -134.018,Y -46.5189,Z 175,A -158.6463,B 7.3307,C 0.3305,E1 7.1866,E2 250.8077} C_DIS
LIN {X -135.1576,Y -43.0958,Z 175,A -160.1455,B 7.3308,C 0.3271,E1 7.1853,E2 252.3114} C_DIS
LIN {X -136.2474,Y -39.5174,Z 175,A -161.6463,B 7.331,C 0.3228,E1 7.1841,E2 253.8099} C_DIS
LIN {X -137.1077,Y -36.4191,Z 175,A -162.973,B 7.3311,C 0.3196,E1 7.1831,E2 255.1392} C_DIS
LIN {X -137.9625,Y -33.0342,Z 175,A -164.4375,B 7.3313,C 0.3165,E1 7.1821,E2 256.6098} C_DIS
LIN {X -138.787,Y -29.3831,Z 175,A -165.9271,B 7.3315,C 0.3119,E1 7.1812,E2 258.0954} C_DIS
LIN {X -139.4169,Y -26.2293,Z 175,A -167.2859,B 7.3315,C 0.3091,E1 7.1805,E2 259.461} C_DIS
LIN {X -140.0401,Y -22.6743,Z 175,A -168.9489,B 7.3316,C 0.3077,E1 7.1797,E2 261.1496} C_DIS
Enddeposition()
END
